# B&R Automation Studio project NAINV104C00R8L515F00 (part 21)

#### Act_Link.st - Change By Project
```iecst
(** 2019-03-29 **)
ACTION Act_Link:

	//Ready Receive
	IF p_bLinkNtParamUSWidthChkPrep AND p_bLinkMcParamUSWidthChkEn THEN
		p_bRdyRcv	:= p_bLinkDIUSWidthChkSen;
	ELSE
		p_bRdyRcv	:= TRUE;
	END_IF

	//Receive Complete Signal
	//p_bComplSigOn	:= p_bLeftSen = FALSE;

	IF EDGENEG(p_bLeftSen) THEN
		p_bComplSigOn	:= TRUE;
	END_IF

	IF eStat <> SMEMAActRun THEN
		p_bComplSigOn	:= FALSE;
	END_IF

	//Direction
	p_bDirLToR	:= p_eLinkConvDir = ConvDirLToR OR p_eLinkConvDir = ConvDirLToL;

END_ACTION
```

#### Act_InitLocal.st - Do Not Change!!!
```iecst
(** 2019-03-25 **)
ACTION Act_InitLocal:

	//Input Reference Link To Local Variable
	p_eAct ACCESS ADR(eAct);
	p_udiRstErr ACCESS ADR(udiRstErr);
	p_bPrep ACCESS ADR(bPrep);
	p_bEn ACCESS ADR(bEn);
	p_bDis ACCESS ADR(bDis);
	p_bManual ACCESS ADR(bManual);
	p_tyParam ACCESS ADR(tyParam);
	p_diTransferInTO ACCESS ADR(diTransferInTO);
	p_bDirLToR ACCESS ADR(bDirLToR);
	p_bRdyRcv ACCESS ADR(bRdyRcv);
	p_bLeftSen ACCESS ADR(bLeftSen);
	p_bRightSen ACCESS ADR(bRightSen);
	p_bComplSigOn ACCESS ADR(bComplSigOn);
	p_bUBA ACCESS ADR(bUBA);
	p_bUBAStat ACCESS ADR(bUBAStat);
	p_bTimerEnSen ACCESS ADR(bTimerEnSen);
	p_bTimerEnSenEdge ACCESS ADR(bTimerEnSenEdge);
	p_bVirtualEn ACCESS ADR(bVirtualEn);
	p_bUBAVirtual ACCESS ADR(bUBAVirtual);
	p_bUBAStatVirtual ACCESS ADR(bUBAStatVirtual);
	p_tRstDlyTm ACCESS ADR(tRstDlyTm);
	p_tSigInChkTm ACCESS ADR(tSigInChkTm);
	p_sProgNm ACCESS ADR(sProgNm);
	p_bNtSettingsLoadDone ACCESS ADR(bNtSettingsLoadDone);

END_ACTION
```

#### Act_Initial.st - Do Not Change!!!
```iecst
(** 2019-03-22 **)
ACTION Act_Initial:

	//Initial
	sStatTxt	:= a_sStatText[eStat];

	fbSMEMA_Std.tRstDlyTm	:= p_tRstDlyTm;
	fbSMEMA_Std(bEn := FALSE);

	fbSMEMA_9851.tRstDlyTm	:= p_tRstDlyTm;
	fbSMEMA_9851(bEn := FALSE);

	fbTimerDlyTm(IN := FALSE);
	fbTimeTrig(CLK := TRUE);

	fbSigInChk.tSigInChkTm	:= p_tSigInChkTm;

END_ACTION
```

#### Act_Background.st - Do Not Change!!!
```iecst
(** 2019-01-20 **)
ACTION Act_Background:

	fbTimeTrig(CLK := p_bTimerEnSenEdge);

	IF eStat = SMEMAActRun AND (p_bTimerEnSenEdge OR p_bTimerEnSen) THEN
		IF fbTimeTrig.Q = TRUE OR p_bTimerEnSen THEN
			fbTimerDlyTm.IN	:= TRUE;
		END_IF
	ELSE
		fbTimerDlyTm.IN	:= FALSE;
	END_IF

	IF bConvStart = FALSE AND bConvStop = FALSE THEN
		fbTimerDlyTm;

		IF fbTimerDlyTm.Q = TRUE AND eStat = SMEMAActRun THEN
			bTimer		:= TRUE;
			bVirtual	:= FALSE;
		ELSIF p_bVirtualEn = TRUE THEN
			bTimer		:= FALSE;
			bVirtual	:= TRUE;
		ELSE
			bTimer		:= FALSE;
			bVirtual	:= FALSE;
		END_IF
	ELSE
		fbTimerDlyTm(IN := FALSE);
	END_IF

	IF bTimer = TRUE THEN

		fbSigInChk.bNomSig			:= bConvStart = FALSE AND bConvStop = FALSE;
		fbSigInChk.bStatSig			:= FALSE;
		fbSigInChk.bStatSigSetGd	:= FALSE;

	ELSIF bVirtual = TRUE THEN

		fbSigInChk.bNomSig	:= p_bUBAVirtual;

		IF p_tyParam.eSelection = SMEMASelIPC9851Ext THEN
			fbSigInChk.bStatSig			:= p_bUBAStatVirtual;
			fbSigInChk.bStatSigSetGd	:= p_tyParam.bStatSigSetGd;
		ELSE
			fbSigInChk.bStatSig			:= FALSE;
			fbSigInChk.bStatSigSetGd	:= FALSE;
		END_IF

	ELSE

		fbSigInChk.bNomSig	:= p_bUBA;

		IF p_tyParam.eSelection = SMEMASelIPC9851Ext THEN
			fbSigInChk.bStatSig			:= p_bUBAStat;
			fbSigInChk.bStatSigSetGd	:= p_tyParam.bStatSigSetGd;
		ELSE
			fbSigInChk.bStatSig			:= FALSE;
			fbSigInChk.bStatSigSetGd	:= FALSE;
		END_IF

	END_IF

	fbSigInChk;

	bUSRdy		:= fbSigInChk.bSigInValid;
	bUSGdBrdRdy	:= fbSigInChk.bGdBrd;

END_ACTION
```

#### InputRef.var - Do Not Change!!!
```iecst
(*2019-03-25*)
(**)
(*General*)
VAR
	p_eAct : REFERENCE TO eSMEMAAction;
	p_udiRstErr : REFERENCE TO UDINT;
	p_bPrep : REFERENCE TO BOOL;
	p_bEn : REFERENCE TO BOOL;
	p_bDis : REFERENCE TO BOOL;
END_VAR
(**)
(*Configuration*)
VAR
	p_bManual : REFERENCE TO BOOL;
	p_tyParam : REFERENCE TO tySMEMAParam;
	p_diTransferInTO : REFERENCE TO DINT;
	p_bDirLToR : REFERENCE TO BOOL;
	p_bRdyRcv : REFERENCE TO BOOL;
END_VAR
(**)
(*Input*)
VAR
	p_bLeftSen : REFERENCE TO BOOL;
	p_bRightSen : REFERENCE TO BOOL;
	p_bComplSigOn : REFERENCE TO BOOL;
	p_bUBA : REFERENCE TO BOOL;
	p_bUBAStat : REFERENCE TO BOOL;
	p_bTimerEnSen : REFERENCE TO BOOL;
	p_bTimerEnSenEdge : REFERENCE TO BOOL;
	p_bVirtualEn : REFERENCE TO BOOL;
	p_bUBAVirtual : REFERENCE TO BOOL;
	p_bUBAStatVirtual : REFERENCE TO BOOL;
	p_tRstDlyTm : REFERENCE TO TIME;
	p_tSigInChkTm : REFERENCE TO TIME;
	p_sProgNm : REFERENCE TO STRING[15];
	p_bNtSettingsLoadDone : REFERENCE TO BOOL;
END_VAR
```

#### Local.var - Do Not Change!!!
```iecst
(*2019-04-30*)
(**)
(*Local Action, State & Status*)
VAR
	eAct : eSMEMAAction := SMEMAActIdle;
	eStat : eSMEMAAction := SMEMAActIdle;
	eStatus : eFBStatus := Idle;
	udiStatus : UDINT := 0;
	sStatTxt : STRING[200] := '';
	a_sStatText : ARRAY[0..50] OF STRING[200] := ['Idling','Upstream SMEMA Running','Turning On USB Signal','NA','Turning Off USB Signal','NA','Turning On USB Signal','Turning Off USB Signal',43('')];
END_VAR
(**)
(*Local Alarm*)
VAR
	tyAlmData : tyAlmDat;
	a_tyAlmText : ARRAY[10000..10099] OF tyAlmTxt := [(sAlmText:='SMEMA 9851 Transport Time Out While Transporting',sRcyText:='Timeout Expired Before Operation Completed. Reset And Resume Operation.'),(sAlmText:='SMEMA 9851 Transport Time Out After Opposite Machine Transport Finished',sRcyText:='Timeout Expired Before Operation Completed. Reset And Resume Operation.'),(sAlmText:='SMEMA 9851 Transport Time Out After Current Machine Transport Finished',sRcyText:='Timeout Expired Before Operation Completed. Reset And Resume Operation.'),(sAlmText:='SMEMA 9851 Transport Time Out After Both Machine Transport Finished And Waiting Outlet Sensor',sRcyText:='Timeout Expired Before Operation Completed. Reset And Resume Operation.'),(sAlmText:='Standard SMEMA Transport Time Out While Transporting',sRcyText:='Timeout Expired Before Operation Completed. Reset And Resume Operation.'),(sAlmText:='Standard SMEMA Transport Time Out After Opposite Machine Transport Finished',sRcyText:='Timeout Expired Before Operation Completed. Reset And Resume Operation.'),(sAlmText:='Standard SMEMA Transport Time Out After Current Machine Transport Finished',sRcyText:='Timeout Expired Before Operation Completed. Reset And Resume Operation.'),(sAlmText:='Standard SMEMA Transport Time Out After Both Machine Transport Finished And Waiting Outlet Sensor',sRcyText:='Timeout Expired Before Operation Completed. Reset And Resume Operation.'),92((0))];
END_VAR
(**)
(*Local Output*)
VAR
	bUSRdy : BOOL := FALSE;
	bUSGdBrdRdy : BOOL := FALSE;
	bDSRdy : BOOL := FALSE;
	bTransporting : BOOL := FALSE;
	bConvStart : BOOL := FALSE;
	bConvStop : BOOL := FALSE;
	bUSB : BOOL := FALSE;
	bTimer : BOOL;
	bVirtual : BOOL;
END_VAR
(**)
(*Local Input*)
VAR
	udiRstErr : UDINT := 0;
	bPrep : BOOL := TRUE;
	bEn : BOOL := TRUE;
	bDis : BOOL := FALSE;
	bManual : BOOL := FALSE;
	tyParam : tySMEMAParam;
	diTransferInTO : DINT := 20000;
	bDirLToR : BOOL := FALSE;
	bRdyRcv : BOOL := TRUE;
	bLeftSen : BOOL := FALSE;
	bRightSen : BOOL := FALSE;
	bComplSigOn : BOOL := FALSE;
	bUBA : BOOL := FALSE;
	bUBAStat : BOOL := FALSE;
	bTimerEnSen : BOOL;
	bTimerEnSenEdge : BOOL;
	bVirtualEn : BOOL;
	bUBAVirtual : BOOL;
	bUBAStatVirtual : BOOL;
	tRstDlyTm : TIME := T#500ms;
	tSigInChkTm : TIME := T#100ms;
	sProgNm : STRING[15] := 'USSMEMA';
	bNtSettingsLoadDone : BOOL := TRUE;
END_VAR
(**)
(*Local*)
VAR
	bRstErr : BOOL;
	udiRstErrOld : UDINT;
	bInitDone : BOOL;
	bInitialDone : BOOL;
	fbTimerDlyTm : TON := (PT:=T#1s);
	fbTimeTrig : R_TRIG;
	fbSMEMA_Std : fbSMEMAUS_Std;
	fbSMEMA_9851 : fbSMEMAUS_9851;
	fbSigInChk : fbSMEMASigInChk;
	eStatOld : eSMEMAAction := SMEMAActIdle;
	udiModuleNum : UDINT := 2701;
END_VAR
```

### DSSMEMA.var - Change By Project
```iecst
(*2019-03-25*)
(**)
(*Action & State & Status*)
VAR
	p_DSSMEMAStat : UDINT;
	p_DSSMEMAStatus : UDINT;
	p_DSSMEMAStatTxt : UDINT;
END_VAR
(**)
(*Alarm*)
VAR
	p_DSSMEMAAlmData : UDINT;
END_VAR
(**)
(*Output*)
VAR
	p_DSSMEMAUSRdy : UDINT;
	p_DSSMEMAUSGdBrdRdy : UDINT;
	p_DSSMEMADSRdy : UDINT;
	p_DSSMEMATransporting : UDINT;
	p_DSSMEMAConvStart : UDINT;
	p_DSSMEMAConvStop : UDINT;
	p_DSSMEMADBA : UDINT;
	p_DSSMEMADBAStat : UDINT;
	p_DSSMEMATimer : UDINT;
	p_DSSMEMAVirtual : UDINT;
END_VAR
```

### Program Logical/SMEMA/DSSMEMA (IEC) - 1.00.0 - NtSMEMA v5.00.0

#### InputRef.var
```iecst
(*2019-03-25*)
(**)
(*General*)
VAR
	p_eAct : REFERENCE TO eSMEMAAction;
	p_udiRstErr : REFERENCE TO UDINT;
	p_bPrep : REFERENCE TO BOOL;
	p_bEn : REFERENCE TO BOOL;
	p_bDis : REFERENCE TO BOOL;
END_VAR
(**)
(*Configuration*)
VAR
	p_bManual : REFERENCE TO BOOL;
	p_tyParam : REFERENCE TO tySMEMAParam;
	p_bGdBrd : REFERENCE TO BOOL;
	p_diTransferOutTO : REFERENCE TO DINT;
	p_bDirLToR : REFERENCE TO BOOL;
	p_bRdySend : REFERENCE TO BOOL;
END_VAR
(**)
(*Input*)
VAR
	p_bLeftSen : REFERENCE TO BOOL;
	p_bRightSen : REFERENCE TO BOOL;
	p_bComplSigOn : REFERENCE TO BOOL;
	p_bDSB : REFERENCE TO BOOL;
	p_bTimerEnSen : REFERENCE TO BOOL;
	p_bTimerEnSenEdge : REFERENCE TO BOOL;
	p_bVirtualEn : REFERENCE TO BOOL;
	p_bDSBVirtual : REFERENCE TO BOOL;
	p_tRstDlyTm : REFERENCE TO TIME;
	p_tSigInChkTm : REFERENCE TO TIME;
	p_sProgNm : REFERENCE TO STRING[15];
	p_bNtSettingsLoadDone : REFERENCE TO BOOL;
END_VAR
```

#### InputRef_Link.var
```iecst
(*2019-04-09*)
(**)
VAR
	p_bLinkOpsRun : REFERENCE TO BOOL;
END_VAR
(**)
VAR
	p_eLinkConvDir : REFERENCE TO eConvDir;
	p_bLinkNtParamDSWidthChkPrep : REFERENCE TO BOOL;
	p_bLinkMcParamDSWidthChkEn : REFERENCE TO BOOL;
	p_bLinkDIDSWidthChkSen : REFERENCE TO BOOL;
	p_usiLinkMcMod : REFERENCE TO USINT;
END_VAR
```

#### Local.var
```iecst
(*2019-04-30*)
(**)
(*Local Action, State & Status*)
VAR
	eAct : eSMEMAAction := SMEMAActIdle;
	eStat : eSMEMAAction := SMEMAActIdle;
	eStatus : eFBStatus := Idle;
	udiStatus : UDINT := 0;
	sStatTxt : STRING[200] := '';
	a_sStatText : ARRAY[0..50] OF STRING[200] := ['Idling','SMEMA Running','Turning On DBA Signal','Turning On DBA Stat Signal','Turning Off DBA Signal','Turning Off DBA Stat Signal','Turning On All DBA Signal','Turning Off All DBA Signal',43('')];
END_VAR
(**)
(*Local Alarm*)
VAR
	tyAlmData : tyAlmDat;
	a_tyAlmText : ARRAY[10000..10099] OF tyAlmTxt := [(sAlmText:='SMEMA 9851 Transport Time Out While Transporting',sRcyText:='Timeout Expired Before Operation Completed. Reset And Resume Operation.'),(sAlmText:='SMEMA 9851 Transport Time Out After Opposite Machine Transport Finished',sRcyText:='Timeout Expired Before Operation Completed. Reset And Resume Operation.'),(sAlmText:='SMEMA 9851 Transport Time Out After Current Machine Transport Finished',sRcyText:='Timeout Expired Before Operation Completed. Reset And Resume Operation.'),(sAlmText:='SMEMA 9851 Transport Time Out After Both Machine Transport Finished And Waiting Outlet Sensor',sRcyText:='Timeout Expired Before Operation Completed. Reset And Resume Operation.'),(sAlmText:='Standard SMEMA Transport Time Out While Transporting',sRcyText:='Timeout Expired Before Operation Completed. Reset And Resume Operation.'),(sAlmText:='Standard SMEMA Transport Time Out After Opposite Machine Transport Finished',sRcyText:='Timeout Expired Before Operation Completed. Reset And Resume Operation.'),(sAlmText:='Standard SMEMA Transport Time Out After Current Machine Transport Finished',sRcyText:='Timeout Expired Before Operation Completed. Reset And Resume Operation.'),(sAlmText:='Standard SMEMA Transport Time Out After Both Machine Transport Finished And Waiting Outlet Sensor',sRcyText:='Timeout Expired Before Operation Completed. Reset And Resume Operation.'),92((0))];
END_VAR
(**)
(*Local Output*)
VAR
	bUSRdy : BOOL := FALSE;
	bUSGdBrdRdy : BOOL := FALSE;
	bDSRdy : BOOL := FALSE;
	bTransporting : BOOL := FALSE;
	bConvStart : BOOL := FALSE;
	bConvStop : BOOL := FALSE;
	bDBA : BOOL := FALSE;
	bDBAStat : BOOL := FALSE;
	bTimer : BOOL;
	bVirtual : BOOL;
END_VAR
(**)
(*Local Input*)
VAR
	udiRstErr : UDINT := 0;
	bPrep : BOOL := TRUE;
	bEn : BOOL := TRUE;
	bDis : BOOL := FALSE;
	bManual : BOOL := FALSE;
	tyParam : tySMEMAParam;
	bGdBrd : BOOL := TRUE;
	diTransferOutTO : DINT := 20000;
	bDirLToR : BOOL := FALSE;
	bRdySend : BOOL := TRUE;
	bLeftSen : BOOL := FALSE;
	bRightSen : BOOL := FALSE;
	bComplSigOn : BOOL := FALSE;
	bDSB : BOOL := FALSE;
	bTimerEnSen : BOOL;
	bTimerEnSenEdge : BOOL;
	bVirtualEn : BOOL;
	bDSBVirtual : BOOL;
	tRstDlyTm : TIME := T#500ms;
	tSigInChkTm : TIME := T#100ms;
	sProgNm : STRING[15] := 'DSSMEMA';
	bNtSettingsLoadDone : BOOL := TRUE;
END_VAR
(**)
(*Local*)
VAR
	bRstErr : BOOL;
	udiRstErrOld : UDINT;
	bInitDone : BOOL;
	bInitialDone : BOOL;
	fbTimerDlyTm : TON := (PT:=T#1s);
	fbTimeTrig : R_TRIG;
	fbSMEMA_OppFirst : fbSMEMADS_OppFirst;
	fbSMEMA : fbSMEMADS;
	fbSigInChk : fbSMEMASigInChk;
	eStatOld : eSMEMAAction := SMEMAActIdle;
	udiModuleNum : UDINT := 2801;
END_VAR
```

#### Act_Action.st
```iecst
(** 2019-03-25 **)
ACTION Act_Action:

	//Reset Error
	IF (eStatus = Error) AND bRstErr THEN
		p_eAct	:= SMEMAActIdle;
		eStat	:= SMEMAActIdle;
	END_IF

	//Set p_eAct
	IF eStatus = Idle OR eStatus = Busy OR eStatus = Done THEN
		eStat	:= p_eAct;
	END_IF

END_ACTION
```

#### Act_Alarm.st
```iecst
(** 2019-03-25 **)
ACTION Act_Alarm:

	//Error
	IF EDGEPOS(eStatus = Error) THEN

		tyAlmData.sProgNm		:= p_sProgNm;
		tyAlmData.udiCode		:= udiStatus;
		tyAlmData.eSeverity		:= AlmSeverityError;
		tyAlmData.udiRunTime	:= tyAlmData.udiRunTime + 1;
		tyAlmData.bAlm			:= TRUE;
		tyAlmData.udiModuleNum  := udiModuleNum;
		g_sDSSMEMAProgNm		:= p_sProgNm;

		//Get Error Message
		IF tyAlmData.udiCode < 10000 OR tyAlmData.udiCode > 10099 THEN
			tyAlmData.sAlmMsg	:= 'Unknown';
			tyAlmData.sRcyMsg	:= 'Unknown';
		ELSE
			tyAlmData.sAlmMsg	:= a_tyAlmText[tyAlmData.udiCode].sAlmText;
			tyAlmData.sRcyMsg	:= a_tyAlmText[tyAlmData.udiCode].sRcyText;
		END_IF

		sStatTxt	:= tyAlmData.sAlmMsg;

	ELSIF bRstErr AND (tyAlmData.udiCode <> 0) THEN

		tyAlmData.udiCode	:= 0;
		tyAlmData.eSeverity	:= AlmSeverityNA;
		tyAlmData.sAlmMsg	:= '';
		tyAlmData.sRcyMsg	:= '';
		tyAlmData.bAlm			:= FALSE;
		sStatTxt	:= a_sStatText[eStat];

	END_IF

END_ACTION
```

#### Act_Background.st
```iecst
(** 2019-01-20 **)
ACTION Act_Background:

	fbTimeTrig(CLK := p_bTimerEnSenEdge);

	IF eStat = SMEMAActRun AND (p_bTimerEnSenEdge OR p_bTimerEnSen) THEN
		IF fbTimeTrig.Q = TRUE OR p_bTimerEnSen THEN
			fbTimerDlyTm.IN	:= TRUE;
		END_IF
	ELSE
		fbTimerDlyTm.IN	:= FALSE;
	END_IF

	IF bConvStart = FALSE AND bConvStop = FALSE THEN
		fbTimerDlyTm;

		IF fbTimerDlyTm.Q = TRUE AND eStat = SMEMAActRun THEN
			bTimer		:= TRUE;
			bVirtual	:= FALSE;
		ELSIF p_bVirtualEn = TRUE THEN
			bTimer		:= FALSE;
			bVirtual	:= TRUE;
		ELSE
			bTimer		:= FALSE;
			bVirtual	:= FALSE;
		END_IF
	ELSE
		fbTimerDlyTm(IN := FALSE);
	END_IF

	IF bTimer = TRUE THEN

		fbSigInChk.bNomSig			:= bConvStart = FALSE AND bConvStop = FALSE;
		fbSigInChk.bStatSig			:= FALSE;
		fbSigInChk.bStatSigSetGd	:= FALSE;

	ELSIF bVirtual = TRUE THEN

		fbSigInChk.bNomSig			:= p_bDSBVirtual;
		fbSigInChk.bStatSig			:= FALSE;
		fbSigInChk.bStatSigSetGd	:= FALSE;

	ELSE

		fbSigInChk.bNomSig			:= p_bDSB;
		fbSigInChk.bStatSig			:= FALSE;
		fbSigInChk.bStatSigSetGd	:= FALSE;

	END_IF

	fbSigInChk;

	bDSRdy	:= fbSigInChk.bSigInValid;

END_ACTION
```

#### Act_InitGlobal.st
```iecst
(** 2019-04-09 **)
ACTION Act_InitGlobal:

	(* Always Change If Project Change *)

	//Pass Data To Link
	p_bLinkOpsRun ACCESS p_OpsRun;

	p_eLinkConvDir ACCESS p_NtParamProjConvDir;
	p_bLinkNtParamDSWidthChkPrep ACCESS p_NtParamDSWidthChkPrep;
	p_bLinkMcParamDSWidthChkEn ACCESS p_McParamDSWidthChkEn;
	p_bLinkDIDSWidthChkSen ACCESS p_DIDSWidthChkSen;

	p_usiLinkMcMod ACCESS p_ProdRcpCurrRcp0McMod;

	//Pass Data To Internal Use
	p_udiRstErr ACCESS p_RstErrReset;
	p_bManual ACCESS p_UIMnlMod;
	p_tyParam ACCESS p_McParamDSSMEMAParam;
	p_diTransferOutTO ACCESS p_McParamTranOutErrDlyTm;
	p_bLeftSen ACCESS p_DIConvLftSen;
	p_bRightSen ACCESS p_DIConvRgtSen;
	p_bDSB ACCESS p_DIDSB;
	p_bVirtualEn ACCESS p_UIVSMEMADSEn;
	p_bDSBVirtual ACCESS p_UIVSMEMADSB;
	p_tRstDlyTm ACCESS p_NtParamDSSMEMARstDlyTm;
	p_tSigInChkTm ACCESS p_NtParamDSSMEMASigInChkTm;
	p_sProgNm ACCESS p_NtParamDSSMEMAProgNm;
	p_bNtSettingsLoadDone ACCESS p_StartupNtSettingsLoadDone;

//	p_bGdBrd ACCESS p_OpsInvertGdBrd;

	(* Always Change If Project Change *)

END_ACTION
```

#### Act_Initial.st
```iecst
(** 2019-04-27 **)
ACTION Act_Initial:

	//Initial
	sStatTxt	:= a_sStatText[eStat];

	fbSMEMA_OppFirst.tRstDlyTm	:= p_tRstDlyTm;
	fbSMEMA_OppFirst(bEn := FALSE);

	fbSMEMA.tRstDlyTm	:= p_tRstDlyTm;
	fbSMEMA(bEn := FALSE);

	fbTimerDlyTm(IN := FALSE);
	fbTimeTrig(CLK := TRUE);

	fbSigInChk.tSigInChkTm	:= p_tSigInChkTm;

END_ACTION
```

#### Act_InitLocal.st
```iecst
(** 2019-03-25 **)
ACTION Act_InitLocal:

	//Input Reference Link To Local Variable
	p_eAct ACCESS ADR(eAct);
	p_udiRstErr ACCESS ADR(udiRstErr);
	p_bPrep ACCESS ADR(bPrep);
	p_bEn ACCESS ADR(bEn);
	p_bDis ACCESS ADR(bDis);
	p_bManual ACCESS ADR(bManual);
	p_tyParam ACCESS ADR(tyParam);
	p_bGdBrd ACCESS ADR(bGdBrd);
	p_diTransferOutTO ACCESS ADR(diTransferOutTO);
	p_bDirLToR ACCESS ADR(bDirLToR);
	p_bRdySend ACCESS ADR(bRdySend);
	p_bLeftSen ACCESS ADR(bLeftSen);
	p_bRightSen ACCESS ADR(bRightSen);
	p_bComplSigOn ACCESS ADR(bComplSigOn);
	p_bDSB ACCESS ADR(bDSB);
	p_bTimerEnSen ACCESS ADR(bTimerEnSen);
	p_bTimerEnSenEdge ACCESS ADR(bTimerEnSenEdge);
	p_bVirtualEn ACCESS ADR(bVirtualEn);
	p_bDSBVirtual ACCESS ADR(bDSBVirtual);
	p_tRstDlyTm ACCESS ADR(tRstDlyTm);
	p_tSigInChkTm ACCESS ADR(tSigInChkTm);
	p_sProgNm ACCESS ADR(sProgNm);
	p_bNtSettingsLoadDone ACCESS ADR(bNtSettingsLoadDone);

END_ACTION
```

#### Act_Link.st
```iecst
(** 2019-03-29 **)
ACTION Act_Link:

	//Ready Send
	IF p_bLinkNtParamDSWidthChkPrep AND p_bLinkMcParamDSWidthChkEn THEN
		p_bRdySend	:= p_bLinkDIDSWidthChkSen;
	ELSE
		p_bRdySend	:= TRUE;
	END_IF

	//Send Complete Signal
	IF EDGENEG(p_bRightSen) THEN
		p_bComplSigOn	:= TRUE;
	END_IF

	IF eStat <> SMEMAActRun THEN
		p_bComplSigOn	:= FALSE;
	END_IF

	//Direction
	p_bDirLToR	:= p_eLinkConvDir = ConvDirLToR OR p_eLinkConvDir = ConvDirLToL;

	//Good Board Access
	IF p_usiLinkMcMod = 0 AND p_usiLinkMcMod = 1 THEN
		p_bGdBrd ACCESS p_OpsInvertGdBrd;
	ELSE
		p_bGdBrd ACCESS p_OpsInvertGdBrd;
	END_IF

END_ACTION
```

#### Act_LinkAction.st
```iecst
(** 2019-04-09 **)
ACTION Act_LinkAction:

	IF p_bLinkOpsRun = TRUE THEN
		p_eAct ACCESS p_OpsInvertDSSMEMAAct;
	ELSIF p_bManual = TRUE THEN
		p_eAct ACCESS p_UIDSSMEMAAct;
	ELSE
		p_eAct ACCESS ADR(eAct);
	END_IF

END_ACTION
```

#### Act_Main.st
```iecst
(** 2019-04-27 **)
ACTION Act_Main:

	IF eStatOld <> eStat THEN
		fbSMEMA_OppFirst(bEn := FALSE);
		fbSMEMA(bEn := FALSE);

		bTransporting	:= FALSE;
		bConvStart		:= FALSE;
		bConvStop		:= FALSE;
		bUSRdy			:= FALSE;
		bUSGdBrdRdy		:= FALSE;

		IF eStatOld <> SMEMAActIdle
			AND eStatOld <> SMEMAActSetSig
			AND eStatOld <> SMEMAActSetStatSig
			AND eStatOld <> SMEMAActRstSig
			AND eStatOld <> SMEMAActRstStatSig
			AND eStatOld <> SMEMAActSetAllSig
			AND eStatOld <> SMEMAActRstAllSig THEN

			bDBA		:= FALSE;
			bDBAStat	:= FALSE;

		END_IF

		sStatTxt	:= a_sStatText[eStat];

		eStatOld	:= eStat;

		eStatus		:= Busy;
	END_IF

	//Main
	CASE eStat OF

		SMEMAActIdle:
			IF EDGENEG(p_bManual) THEN
				bDBA		:= FALSE;
				bDBAStat	:= FALSE;
			END_IF

			eStatus	:= Idle;

		SMEMAActRun:
			IF eStatus = Idle OR eStatus = Busy THEN

				eStatus	:= Busy;

				IF p_tyParam.eSelection <> SMEMASelStandard THEN

					fbSMEMA.bDSRdy		:= fbSigInChk.bSigInValid;
					fbSMEMA.bRdySend	:= p_bRdySend;
					fbSMEMA.bComplSigOn	:= p_bComplSigOn;

					fbSMEMA.tTimeOut	:= DINT_TO_TIME(p_diTransferOutTO);
					fbSMEMA(bEn := TRUE);

					bTransporting	:= fbSMEMA.bTransporting;
					bConvStart		:= fbSMEMA.bConvStart;
					bConvStop		:= fbSMEMA.bConvStop;
					bDBA			:= fbSMEMA.bSigToDS AND (bTimer = FALSE) AND (bVirtual = FALSE);
					bDBAStat		:= (fbSMEMA.bSigToDS) AND (fSMEMASigStatOut(p_tyParam.bStatSigSetGd, p_bGdBrd)) AND (p_tyParam.eSelection = SMEMASelIPC9851Ext);

					bUSRdy			:= fbSMEMA.bSigToDS;
					bUSGdBrdRdy		:= p_bGdBrd;

					IF fbSMEMA.udiStatus = 0 THEN
						eStatus	:= Done;
					ELSIF fbSMEMA.udiStatus < 65534 THEN
						eStatus		:= Error;

						IF fbSMEMA.udiStatus = 1200 THEN
							udiStatus	:= 10000;	//SMEMA 9851 Transport Time Out While Transporting
						ELSIF fbSMEMA.udiStatus = 1201 THEN
							udiStatus	:= 10001;	//SMEMA 9851 Transport Time Out After Opposite Machine Transport Finished
						ELSIF fbSMEMA.udiStatus = 1202 THEN
							udiStatus	:= 10002;	//SMEMA 9851 Transport Time Out After Current Machine Transport Finished
						ELSIF fbSMEMA.udiStatus = 1203 THEN
							udiStatus	:= 10003;	//SMEMA 9851 Transport Time Out After Both Machine Transport Finished And Waiting Outlet Sensor
						ELSE
							udiStatus	:= fbSMEMA.udiStatus;
						END_IF
					END_IF

				ELSE

					fbSMEMA_OppFirst.bDSRdy			:= fbSigInChk.bSigInValid;
					fbSMEMA_OppFirst.bRdySend		:= p_bRdySend;
					fbSMEMA_OppFirst.bComplSigOn	:= p_bComplSigOn;

					fbSMEMA_OppFirst.tTimeOut	:= DINT_TO_TIME(p_diTransferOutTO);
					fbSMEMA_OppFirst(bEn := TRUE);

					bTransporting	:= fbSMEMA_OppFirst.bTransporting;
					bConvStart		:= fbSMEMA_OppFirst.bConvStart;
					bConvStop		:= fbSMEMA_OppFirst.bConvStop;
					bDBA			:= fbSMEMA_OppFirst.bSigToDS AND (bTimer = FALSE) AND (bVirtual = FALSE);
					bDBAStat		:= (fbSMEMA_OppFirst.bSigToDS) AND (fSMEMASigStatOut(p_tyParam.bStatSigSetGd, p_bGdBrd)) AND (p_tyParam.eSelection = SMEMASelIPC9851Ext);

					bUSRdy			:= fbSMEMA_OppFirst.bSigToDS;
					bUSGdBrdRdy		:= p_bGdBrd;

					IF fbSMEMA_OppFirst.udiStatus = 0 THEN
						eStatus	:= Done;
					ELSIF fbSMEMA_OppFirst.udiStatus < 65534 THEN
						eStatus		:= Error;

						IF fbSMEMA_OppFirst.udiStatus = 1200 THEN
							udiStatus	:= 10004;	//Standard SMEMA Transport Time Out While Transporting
						ELSIF fbSMEMA_OppFirst.udiStatus = 1201 THEN
							udiStatus	:= 10005;	//Standard SMEMA Transport Time Out After Opposite Machine Transport Finished
						ELSIF fbSMEMA_OppFirst.udiStatus = 1202 THEN
							udiStatus	:= 10006;	//Standard SMEMA Transport Time Out After Current Machine Transport Finished
						ELSIF fbSMEMA_OppFirst.udiStatus = 1203 THEN
							udiStatus	:= 10007;	//Standard SMEMA Transport Time Out After Both Machine Transport Finished And Waiting Outlet Sensor
						ELSE
							udiStatus	:= fbSMEMA_OppFirst.udiStatus;
						END_IF
					END_IF

				END_IF

			END_IF

		SMEMAActSetSig:
			IF eStatus = Idle OR eStatus = Busy THEN

				//Reset
				fbSMEMA_OppFirst(bEn := FALSE);
				fbSMEMA(bEn := FALSE);

				bConvStart	:= FALSE;
				bConvStop	:= FALSE;

				bDBA	:= TRUE;
				eStatus	:= Done;

			END_IF

		SMEMAActSetStatSig:
			IF eStatus = Idle OR eStatus = Busy THEN

				//Reset
				fbSMEMA_OppFirst(bEn := FALSE);
				fbSMEMA(bEn := FALSE);

				bConvStart	:= FALSE;
				bConvStop	:= FALSE;

				bDBAStat	:= TRUE;
				eStatus		:= Done;

			END_IF

		SMEMAActRstSig:
			IF eStatus = Idle OR eStatus = Busy THEN

				//Reset
				fbSMEMA_OppFirst(bEn := FALSE);
				fbSMEMA(bEn := FALSE);

				bConvStart	:= FALSE;
				bConvStop	:= FALSE;

				bDBA	:= FALSE;
				eStatus	:= Done;

			END_IF

		SMEMAActRstStatSig:
			IF eStatus = Idle OR eStatus = Busy THEN

				//Reset
				fbSMEMA_OppFirst(bEn := FALSE);
				fbSMEMA(bEn := FALSE);

				bConvStart	:= FALSE;
				bConvStop	:= FALSE;

				bDBAStat	:= FALSE;
				eStatus		:= Done;

			END_IF

		SMEMAActSetAllSig:
			IF eStatus = Idle OR eStatus = Busy THEN

				//Reset
				fbSMEMA_OppFirst(bEn := FALSE);
				fbSMEMA(bEn := FALSE);

				bConvStart	:= FALSE;
				bConvStop	:= FALSE;

				bDBA		:= TRUE;
				bDBAStat	:= TRUE;
				eStatus		:= Done;

			END_IF

		SMEMAActRstAllSig:
			IF eStatus = Idle OR eStatus = Busy THEN

				//Reset
				fbSMEMA_OppFirst(bEn := FALSE);
				fbSMEMA(bEn := FALSE);

				bConvStart	:= FALSE;
				bConvStop	:= FALSE;

				bDBA		:= FALSE;
				bDBAStat	:= FALSE;
				eStatus		:= Done;

			END_IF

	END_CASE

END_ACTION
```

#### Init.st
```iecst
(** 2019-03-25 **)
PROGRAM _INIT

	(* Always Change If Project Change *)

	//Pass Address To Global Address For External Use
	//Action, State & Status
	p_DSSMEMAStat		:= ADR(eStat);
	p_DSSMEMAStatus		:= ADR(eStatus);
	p_DSSMEMAStatTxt	:= ADR(sStatTxt);

	//Alarm
	p_DSSMEMAAlmData	:= ADR(tyAlmData);

	//Output
	p_DSSMEMAUSRdy			:= ADR(bUSRdy);
	p_DSSMEMAUSGdBrdRdy		:= ADR(bUSGdBrdRdy);
	p_DSSMEMADSRdy			:= ADR(bDSRdy);
	p_DSSMEMATransporting	:= ADR(bTransporting);
	p_DSSMEMAConvStart		:= ADR(bConvStart);
	p_DSSMEMAConvStop		:= ADR(bConvStop);
	p_DSSMEMADBA			:= ADR(bDBA);
	p_DSSMEMADBAStat		:= ADR(bDBAStat);
	p_DSSMEMATimer			:= ADR(bTimer);
	p_DSSMEMAVirtual		:= ADR(bVirtual);

	(* Always Change If Project Change *)

END_PROGRAM
```

### USSMEMA2.var - Change By Project
```iecst
(*2019-03-25*)
(**)
(*Action & State & Status*)
VAR
	p_USSMEMA2Stat : UDINT;
	p_USSMEMA2Status : UDINT;
	p_USSMEMA2StatTxt : UDINT;
END_VAR
(**)
(*Alarm*)
VAR
	p_USSMEMA2AlmData : UDINT;
END_VAR
(**)
(*Output*)
VAR
	p_USSMEMA2USRdy : UDINT;
	p_USSMEMA2USGdBrdRdy : UDINT;
	p_USSMEMA2DSRdy : UDINT;
	p_USSMEMA2Transporting : UDINT;
	p_USSMEMA2ConvStart : UDINT;
	p_USSMEMA2ConvStop : UDINT;
	p_USSMEMA2USB : UDINT;
	p_USSMEMA2Timer : UDINT;
	p_USSMEMA2Virtual : UDINT;
END_VAR
```

### Program Logical/SMEMA/USSMEMA2 (IEC, version 1.00.0) - 1.00.0 - NtSMEMA v5.00.0

#### Init.st - Change By Project
```iecst
(** 2019-03-25 **)
PROGRAM _INIT

	(* Always Change If Project Change *)

	//Pass Address To Global Address For External Use
	//Action, State & Status
	p_USSMEMA2Stat		:= ADR(eStat);
	p_USSMEMA2Status		:= ADR(eStatus);
	p_USSMEMA2StatTxt	:= ADR(sStatTxt);

	//Alarm
	p_USSMEMA2AlmData	:= ADR(tyAlmData);

	//Output
	p_USSMEMA2USRdy			:= ADR(bUSRdy);
	p_USSMEMA2USGdBrdRdy	:= ADR(bUSGdBrdRdy);
	p_USSMEMA2DSRdy			:= ADR(bDSRdy);
	p_USSMEMA2Transporting	:= ADR(bTransporting);
	p_USSMEMA2ConvStart		:= ADR(bConvStart);
	p_USSMEMA2ConvStop		:= ADR(bConvStop);
	p_USSMEMA2USB			:= ADR(bUSB);
	p_USSMEMA2Timer			:= ADR(bTimer);
	p_USSMEMA2Virtual		:= ADR(bVirtual);

	(* Always Change If Project Change *)

END_PROGRAM
```

#### Act_InitGlobal.st - Change By Project
```iecst
(** 2019-04-09 **)
ACTION Act_InitGlobal:

	(* Always Change If Project Change *)

	//Pass Data To Link
	p_bLinkOpsRun ACCESS p_OpsRun;

	p_eLinkConvDir ACCESS p_NtParamProjConvDir;
	p_bLinkNtParamUSWidthChkPrep ACCESS p_NtParamUSWidthChkPrep;
	p_bLinkMcParamUSWidthChkEn ACCESS p_McParamUSWidthChkEn;
	p_bLinkDIUSWidthChkSen ACCESS p_DIUSWidthChkSen;
	p_usiLinkMcMod ACCESS p_ProdRcpCurrRcp0McMod;

	//Pass Data To Internal Use
	p_udiRstErr ACCESS p_RstErrReset;
	p_bManual ACCESS p_UIMnlMod;
	p_tyParam ACCESS p_McParamUSSMEMA2Param;
	p_diTransferInTO ACCESS p_McParamTranInErrDlyTm;
	p_bLeftSen ACCESS p_DIConvLftSen;
	p_bRightSen ACCESS p_DIConvRgtSen;
	p_bUBA ACCESS p_DIUBA2;
	p_bUBAStat ACCESS p_DIUBAStat2;
	p_bVirtualEn ACCESS p_UIVSMEMAUS2En;
	p_bUBAVirtual ACCESS p_UIVSMEMAUBA2;
	p_bUBAStatVirtual ACCESS p_UIVSMEMAUBAStat2;
	p_tRstDlyTm ACCESS p_NtParamUSSMEMA2RstDlyTm;
	p_tSigInChkTm ACCESS p_NtParamUSSMEMA2SigInChkTm;
	p_sProgNm ACCESS p_NtParamUSSMEMA2ProgNm;
	p_bNtSettingsLoadDone ACCESS p_StartupNtSettingsLoadDone;

	(* Always Change If Project Change *)

END_ACTION
```

#### InputRef_Link.var - Change By Project
```iecst
(*2019-04-09*)
(**)
VAR
	p_bLinkOpsRun : REFERENCE TO BOOL;
END_VAR
(**)
VAR
	p_eLinkConvDir : REFERENCE TO eConvDir;
	p_bLinkNtParamUSWidthChkPrep : REFERENCE TO BOOL;
	p_bLinkMcParamUSWidthChkEn : REFERENCE TO BOOL;
	p_bLinkDIUSWidthChkSen : REFERENCE TO BOOL;
	p_usiLinkMcMod : REFERENCE TO USINT;
END_VAR
```

#### Act_LinkAction.st - Change By Project
```iecst
(** 2019-04-09 **)
ACTION Act_LinkAction:

	IF p_bLinkOpsRun = TRUE THEN
		p_eAct ACCESS p_OpsInvertUSSMEMA2Act;
	ELSIF p_bManual = TRUE THEN
		p_eAct ACCESS p_UIUSSMEMA2Act;
	ELSE
		p_eAct ACCESS ADR(eAct);
	END_IF

END_ACTION
```

#### Act_Link.st - Change By Project
```iecst
(** 2019-03-29 **)
ACTION Act_Link:

	//Ready Receive
	IF p_bLinkNtParamUSWidthChkPrep AND p_bLinkMcParamUSWidthChkEn THEN
		p_bRdyRcv	:= p_bLinkDIUSWidthChkSen;
	ELSE
		p_bRdyRcv	:= TRUE;
	END_IF

	//Receive Complete Signal
	//p_bComplSigOn	:= p_bLeftSen = FALSE;

	IF EDGENEG(p_bRightSen) THEN
		p_bComplSigOn	:= TRUE;
	END_IF

	IF eStat <> SMEMAActRun THEN
		p_bComplSigOn	:= FALSE;
	END_IF

	//Direction
	//	p_bDirLToR	:= p_eLinkConvDir = ConvDirLToR OR p_eLinkConvDir = ConvDirLToL;

		p_bDirLToR	:= p_eLinkConvDir = ConvDirRToL OR p_eLinkConvDir = ConvDirRToR;

END_ACTION
```

#### Cyclic.st - Do Not Change!!!
```iecst
(** 2019-03-29 **)
PROGRAM _CYCLIC

	IF bInitDone = FALSE THEN
		bInitDone	:= TRUE;

		Act_InitLocal;
		Act_InitGlobal;

	ELSIF bInitialDone = FALSE THEN
		IF p_bNtSettingsLoadDone = TRUE THEN
			bInitialDone	:= TRUE;

			Act_Initial;
		END_IF

	ELSE

		Act_RstErr;
		Act_LinkAction;
		Act_Action;
		Act_LinkEn;

		IF (p_bPrep = TRUE) AND (p_bEn = TRUE) AND (p_bDis = FALSE) THEN
			Act_Link;
			Act_Background;
			Act_Main;
		ELSE
			IF eStat <> SMEMAActIdle THEN
				eStatus	:= Done;
			ELSE
				eStatus	:= Idle;
			END_IF
		END_IF

		Act_Alarm;

	END_IF

END_PROGRAM
```

#### Act_RstErr.st - Do Not Change!!!
```iecst
(** 2018-12-08 **)
ACTION Act_RstErr:

	IF p_udiRstErr <> udiRstErrOld THEN
		bRstErr			:= TRUE;
		udiRstErrOld	:= p_udiRstErr;
	ELSE
		bRstErr			:= FALSE;
	END_IF

END_ACTION
```

#### Act_Action.st - Do Not Change!!!
```iecst
(** 2019-03-25 **)
ACTION Act_Action:

	//Reset Error
	IF (eStatus = Error) AND bRstErr THEN
		p_eAct	:= SMEMAActIdle;
		eStat	:= SMEMAActIdle;
	END_IF

	//Set p_eAct
	IF eStatus = Idle OR eStatus = Busy OR eStatus = Done THEN
		eStat	:= p_eAct;
	END_IF

END_ACTION
```

#### Act_Main.st - Do Not Change!!!
```iecst
(** 2019-03-22 **)
ACTION Act_Main:

	IF eStatOld <> eStat THEN
		fbSMEMA_Std(bEn := FALSE);
		fbSMEMA_9851(bEn := FALSE);

		bTransporting	:= FALSE;
		bConvStart		:= FALSE;
		bConvStop		:= FALSE;
		bDSRdy			:= FALSE;

		IF eStatOld <> SMEMAActIdle
			AND eStatOld <> SMEMAActSetSig
			AND eStatOld <> SMEMAActSetStatSig
			AND eStatOld <> SMEMAActRstSig
			AND eStatOld <> SMEMAActRstStatSig
			AND eStatOld <> SMEMAActSetAllSig
			AND eStatOld <> SMEMAActRstAllSig THEN

			bUSB	:= FALSE;

		END_IF

		sStatTxt	:= a_sStatText[eStat];

		eStatOld	:= eStat;

		eStatus		:= Busy;
	END_IF

	//Main
	CASE eStat OF

		SMEMAActIdle:
			IF EDGENEG(p_bManual) THEN
				bUSB	:= FALSE;
			END_IF

			eStatus	:= Idle;

		SMEMAActRun:
			IF eStatus = Idle OR eStatus = Busy THEN

				eStatus	:= Busy;

				IF p_tyParam.eSelection <> SMEMASelStandard THEN

					fbSMEMA_9851.bUSRdy			:= fbSigInChk.bSigInValid;
					fbSMEMA_9851.bRdyRcv		:= p_bRdyRcv;
					fbSMEMA_9851.bComplSigOn	:= p_bComplSigOn;

					IF p_bDirLToR = TRUE THEN

						fbSMEMA_9851.bInletSen		:= p_bLeftSen;
						fbSMEMA_9851.bOutletSen		:= p_bRightSen;

					ELSE

						fbSMEMA_9851.bInletSen		:= p_bRightSen;
						fbSMEMA_9851.bOutletSen		:= p_bLeftSen;

					END_IF

					fbSMEMA_9851.tTimeOut	:= DINT_TO_TIME(p_diTransferInTO);
					fbSMEMA_9851(bEn := TRUE);

					bTransporting	:= fbSMEMA_9851.bTransporting;
					bConvStart		:= fbSMEMA_9851.bConvStart;
					bConvStop		:= fbSMEMA_9851.bConvStop;
					bUSB			:= fbSMEMA_9851.bSigToUS AND (bTimer = FALSE) AND (bVirtual = FALSE);
					bDSRdy			:= fbSMEMA_9851.bSigToUS;

					IF fbSMEMA_9851.udiStatus = 0 THEN
						eStatus	:= Done;
					ELSIF fbSMEMA_9851.udiStatus < 65534 THEN
						eStatus		:= Error;

						IF fbSMEMA_9851.udiStatus = 1200 THEN
							udiStatus	:= 10000;	//SMEMA 9851 Transport Time Out While Transporting
						ELSIF fbSMEMA_9851.udiStatus = 1201 THEN
							udiStatus	:= 10001;	//SMEMA 9851 Transport Time Out After Opposite Machine Transport Finished
						ELSIF fbSMEMA_9851.udiStatus = 1202 THEN
							udiStatus	:= 10002;	//SMEMA 9851 Transport Time Out After Current Machine Transport Finished
						ELSIF fbSMEMA_9851.udiStatus = 1203 THEN
							udiStatus	:= 10003;	//SMEMA 9851 Transport Time Out After Both Machine Transport Finished And Waiting Outlet Sensor
						ELSE
							udiStatus	:= fbSMEMA_9851.udiStatus;
						END_IF
					END_IF

				ELSE

					fbSMEMA_Std.bUSRdy		:= fbSigInChk.bSigInValid;
					fbSMEMA_Std.bRdyRcv		:= p_bRdyRcv;
					fbSMEMA_Std.bComplSigOn	:= p_bComplSigOn;

					IF p_bDirLToR = TRUE THEN

						fbSMEMA_Std.bInletSen	:= p_bLeftSen;
						fbSMEMA_Std.bOutletSen	:= p_bRightSen;

					ELSE

						fbSMEMA_Std.bInletSen	:= p_bRightSen;
						fbSMEMA_Std.bOutletSen	:= p_bLeftSen;

					END_IF

					fbSMEMA_Std.tTimeOut	:= DINT_TO_TIME(p_diTransferInTO);
					fbSMEMA_Std(bEn := TRUE);

					bTransporting	:= fbSMEMA_Std.bTransporting;
					bConvStart		:= fbSMEMA_Std.bConvStart;
					bConvStop		:= fbSMEMA_Std.bConvStop;
					bUSB			:= fbSMEMA_Std.bSigToUS AND (bTimer = FALSE) AND (bVirtual = FALSE);
					bDSRdy			:= fbSMEMA_Std.bSigToUS;

					IF fbSMEMA_Std.udiStatus = 0 THEN
						eStatus	:= Done;
					ELSIF fbSMEMA_Std.udiStatus < 65534 THEN
						eStatus		:= Error;

						IF fbSMEMA_Std.udiStatus = 1200 THEN
							udiStatus	:= 10004;	//Standard SMEMA Transport Time Out While Transporting
						ELSIF fbSMEMA_Std.udiStatus = 1201 THEN
							udiStatus	:= 10005;	//Standard SMEMA Transport Time Out After Opposite Machine Transport Finished
						ELSIF fbSMEMA_Std.udiStatus = 1202 THEN
							udiStatus	:= 10006;	//Standard SMEMA Transport Time Out After Current Machine Transport Finished
						ELSIF fbSMEMA_Std.udiStatus = 1203 THEN
							udiStatus	:= 10007;	//Standard SMEMA Transport Time Out After Both Machine Transport Finished And Waiting Outlet Sensor
						ELSE
							udiStatus	:= fbSMEMA_Std.udiStatus;
						END_IF
					END_IF

				END_IF

			END_IF

		SMEMAActSetSig:
			IF eStatus = Idle OR eStatus = Busy THEN

				//Reset
				fbSMEMA_Std(bEn := FALSE);
				fbSMEMA_9851(bEn := FALSE);

				bConvStart	:= FALSE;
				bConvStop	:= FALSE;

				bUSB	:= TRUE;
				eStatus	:= Done;

			END_IF

		SMEMAActSetStatSig:
			IF eStatus = Idle OR eStatus = Busy THEN

				//Reset
				fbSMEMA_Std(bEn := FALSE);
				fbSMEMA_9851(bEn := FALSE);

				bConvStart	:= FALSE;
				bConvStop	:= FALSE;

				eStatus	:= Done;

			END_IF

		SMEMAActRstSig:
			IF eStatus = Idle OR eStatus = Busy THEN

				//Reset
				fbSMEMA_Std(bEn := FALSE);
				fbSMEMA_9851(bEn := FALSE);

				bConvStart	:= FALSE;
				bConvStop	:= FALSE;

				bUSB	:= FALSE;
				eStatus	:= Done;

			END_IF

		SMEMAActRstStatSig:
			IF eStatus = Idle OR eStatus = Busy THEN

				//Reset
				fbSMEMA_Std(bEn := FALSE);
				fbSMEMA_9851(bEn := FALSE);

				bConvStart	:= FALSE;
				bConvStop	:= FALSE;

				eStatus	:= Done;

			END_IF

		SMEMAActSetAllSig:
			IF eStatus = Idle OR eStatus = Busy THEN

				//Reset
				fbSMEMA_Std(bEn := FALSE);
				fbSMEMA_9851(bEn := FALSE);

				bConvStart	:= FALSE;
				bConvStop	:= FALSE;

				bUSB	:= TRUE;
				eStatus	:= Done;

			END_IF

		SMEMAActRstAllSig:
			IF eStatus = Idle OR eStatus = Busy THEN

				//Reset
				fbSMEMA_Std(bEn := FALSE);
				fbSMEMA_9851(bEn := FALSE);

				bConvStart	:= FALSE;
				bConvStop	:= FALSE;

				bUSB	:= FALSE;
				eStatus	:= Done;

			END_IF

	END_CASE

END_ACTION
```

#### Act_Alarm.st - Do Not Change!!!
```iecst
(** 2019-03-25 **)
ACTION Act_Alarm:

	//Error
	IF EDGEPOS(eStatus = Error) THEN

		tyAlmData.sProgNm		:= p_sProgNm;
		tyAlmData.udiCode		:= udiStatus;
		tyAlmData.eSeverity		:= AlmSeverityError;
		tyAlmData.udiRunTime	:= tyAlmData.udiRunTime + 1;
		tyAlmData.bAlm			:= TRUE;
		tyAlmData.udiModuleNum  := udiModuleNum;
		g_sUSSMEMAProgNm		:= p_sProgNm;

		//Get Error Message
		IF tyAlmData.udiCode < 10000 OR tyAlmData.udiCode > 10099 THEN
			tyAlmData.sAlmMsg	:= 'Unknown';
			tyAlmData.sRcyMsg	:= 'Unknown';
		ELSE
			tyAlmData.sAlmMsg	:= a_tyAlmText[tyAlmData.udiCode].sAlmText;
			tyAlmData.sRcyMsg	:= a_tyAlmText[tyAlmData.udiCode].sRcyText;
		END_IF

		sStatTxt	:= tyAlmData.sAlmMsg;

	ELSIF bRstErr AND (tyAlmData.udiCode <> 0) THEN

		tyAlmData.udiCode	:= 0;
		tyAlmData.eSeverity	:= AlmSeverityNA;
		tyAlmData.sAlmMsg	:= '';
		tyAlmData.sRcyMsg	:= '';
		tyAlmData.bAlm			:= FALSE;

		sStatTxt	:= a_sStatText[eStat];

	END_IF

END_ACTION
```

#### Local.var - Do Not Change!!!
```iecst
(*2019-04-30*)
(**)
(*Local Action, State & Status*)
VAR
	eAct : eSMEMAAction := SMEMAActIdle;
	eStat : eSMEMAAction := SMEMAActIdle;
	eStatus : eFBStatus := Idle;
	udiStatus : UDINT := 0;
	sStatTxt : STRING[200] := '';
	a_sStatText : ARRAY[0..50] OF STRING[200] := ['Idling','Upstream SMEMA Running','Turning On USB Signal','NA','Turning Off USB Signal','NA','Turning On USB Signal','Turning Off USB Signal',43('')];
END_VAR
(**)
(*Local Alarm*)
VAR
	tyAlmData : tyAlmDat;
	a_tyAlmText : ARRAY[10000..10099] OF tyAlmTxt := [(sAlmText:='SMEMA 9851 Transport Time Out While Transporting',sRcyText:='Timeout Expired Before Operation Completed. Reset And Resume Operation.'),(sAlmText:='SMEMA 9851 Transport Time Out After Opposite Machine Transport Finished',sRcyText:='Timeout Expired Before Operation Completed. Reset And Resume Operation.'),(sAlmText:='SMEMA 9851 Transport Time Out After Current Machine Transport Finished',sRcyText:='Timeout Expired Before Operation Completed. Reset And Resume Operation.'),(sAlmText:='SMEMA 9851 Transport Time Out After Both Machine Transport Finished And Waiting Outlet Sensor',sRcyText:='Timeout Expired Before Operation Completed. Reset And Resume Operation.'),(sAlmText:='Standard SMEMA Transport Time Out While Transporting',sRcyText:='Timeout Expired Before Operation Completed. Reset And Resume Operation.'),(sAlmText:='Standard SMEMA Transport Time Out After Opposite Machine Transport Finished',sRcyText:='Timeout Expired Before Operation Completed. Reset And Resume Operation.'),(sAlmText:='Standard SMEMA Transport Time Out After Current Machine Transport Finished',sRcyText:='Timeout Expired Before Operation Completed. Reset And Resume Operation.'),(sAlmText:='Standard SMEMA Transport Time Out After Both Machine Transport Finished And Waiting Outlet Sensor',sRcyText:='Timeout Expired Before Operation Completed. Reset And Resume Operation.'),92((0))];
END_VAR
(**)
(*Local Output*)
VAR
	bUSRdy : BOOL := FALSE;
	bUSGdBrdRdy : BOOL := FALSE;
	bDSRdy : BOOL := FALSE;
	bTransporting : BOOL := FALSE;
	bConvStart : BOOL := FALSE;
	bConvStop : BOOL := FALSE;
	bUSB : BOOL := FALSE;
	bTimer : BOOL;
	bVirtual : BOOL;
END_VAR
(**)
(*Local Input*)
VAR
	udiRstErr : UDINT := 0;
	bPrep : BOOL := TRUE;
	bEn : BOOL := TRUE;
	bDis : BOOL := FALSE;
	bManual : BOOL := FALSE;
	tyParam : tySMEMAParam;
	diTransferInTO : DINT := 20000;
	bDirLToR : BOOL := FALSE;
	bRdyRcv : BOOL := TRUE;
	bLeftSen : BOOL := FALSE;
	bRightSen : BOOL := FALSE;
	bComplSigOn : BOOL := FALSE;
	bUBA : BOOL := FALSE;
	bUBAStat : BOOL := FALSE;
	bTimerEnSen : BOOL;
	bTimerEnSenEdge : BOOL;
	bVirtualEn : BOOL;
	bUBAVirtual : BOOL;
	bUBAStatVirtual : BOOL;
	tRstDlyTm : TIME := T#500ms;
	tSigInChkTm : TIME := T#100ms;
	sProgNm : STRING[15] := 'USSMEMA2';
	bNtSettingsLoadDone : BOOL := TRUE;
END_VAR
(**)
(*Local*)
VAR
	bRstErr : BOOL;
	udiRstErrOld : UDINT;
	bInitDone : BOOL;
	bInitialDone : BOOL;
	fbTimerDlyTm : TON := (PT:=T#1s);
	fbTimeTrig : R_TRIG;
	fbSMEMA_Std : fbSMEMAUS_Std;
	fbSMEMA_9851 : fbSMEMAUS_9851;
	fbSigInChk : fbSMEMASigInChk;
	eStatOld : eSMEMAAction := SMEMAActIdle;
	udiModuleNum : UDINT := 2701;
END_VAR
```

### Pneu.typ - Do Not Change!!!
```iecst
(*2018-12-11*)
(**)
(*Action*)

TYPE
	ePneuAction :
		(
		PneuActIdle,
		PneuActSetAll,
		PneuActRstAll,
		PneuActSetExt,
		PneuActSetRet,
		PneuActExt,
		PneuActRet,
		PneuActExtSenToMidSen,
		PneuActMidSenToRetSen,
		PneuActRetSenToMidSen,
		PneuActMidSenToExtSen
		);
END_TYPE

(**)

TYPE
	eClampType :
		(
		ClampNoRS := 0,
		ThreeClampsWithRS := 1
		);
END_TYPE
```

### PneuNoSenStopper.var - Change By Project
```iecst
(*2019-03-25*)
(**)
(*Action & State & Status*)
VAR
	p_PneuNoSenStopperStat : UDINT;
	p_PneuNoSenStopperStatus : UDINT;
	p_PneuNoSenStopperStatTxt : UDINT;
END_VAR
(**)
(*Alarm*)
VAR
	p_PneuNoSenStopperAlmData : UDINT;
END_VAR
(**)
(*Output*)
VAR
	p_PneuNoSenStopperExtCtrl : UDINT;
	p_PneuNoSenStopperRetCtrl : UDINT;
	p_PneuNoSenStopperTwoCtrlOut : UDINT;
	p_PneuNoSenStopperExtended : UDINT;
	p_PneuNoSenStopperRetracted : UDINT;
END_VAR
```

### Program Logical/Pneu/PneuNoSenStopper (IEC, version 1.00.0) - 1.00.0 - NtPneu v5.00.0

#### Init.st - Change By Project
```iecst
(** 2019-03-25 **)
PROGRAM _INIT

	(* Always Change If Project Change *)

	//Pass Address To Global Address For External Use
	//Action, State & Status
	p_PneuNoSenStopperStat			:= ADR(eStat);
	p_PneuNoSenStopperStatus		:= ADR(eStatus);
	p_PneuNoSenStopperStatTxt		:= ADR(sStatTxt);

	//Alarm
	p_PneuNoSenStopperAlmData		:= ADR(tyAlmData);

	//Output
	p_PneuNoSenStopperExtCtrl		:= ADR(bExtCtrl);
	p_PneuNoSenStopperRetCtrl		:= ADR(bRetCtrl);
	p_PneuNoSenStopperTwoCtrlOut	:= ADR(bTwoCtrlOut);
	p_PneuNoSenStopperExtended		:= ADR(bExtended);
	p_PneuNoSenStopperRetracted		:= ADR(bRetracted);

	(* Always Change If Project Change *)

END_PROGRAM
```

#### Act_InitGlobal.st - Change By Project
```iecst
(** 2019-04-09 **)
ACTION Act_InitGlobal:

	(* Always Change If Project Change *)

	//Pass Data To Link
	p_bLinkOpsRun ACCESS p_OpsRun;
	p_bLinkOpsSimu ACCESS p_SimuRun;

	p_bLinkDISafetyRlySig ACCESS p_DISafetyRlySig;

	//Pass Data To Internal Use
	p_udiRstErr ACCESS p_RstErrReset;
	p_bPrep ACCESS p_NtParamProjStopperPrep;
	p_bDis ACCESS p_McParamStopperDis;
	p_bManual ACCESS p_UIMnlMod;
	p_bTwoCtrlIn ACCESS p_NtParamStopperTwoCtrlIn;
	p_sProgNm ACCESS p_NtParamStopperProgNm;
	p_tExtDlyTm ACCESS p_NtParamStopperExtDlyTm;
	p_tRetDlyTm ACCESS p_NtParamStopperRetDlyTm;
	p_bNtSettingsLoadDone ACCESS p_StartupNtSettingsLoadDone;

	(* Always Change If Project Change *)

END_ACTION
```

#### Act_LinkAction.st - Change By Project
```iecst
(** 2019-04-09 **)
ACTION Act_LinkAction:

	IF p_bLinkOpsRun = TRUE THEN
		p_eAct ACCESS p_OpsInvertStopperAct;
	ELSIF p_bLinkOpsSimu = TRUE THEN
		p_eAct ACCESS p_SimuInvStopperAct;
	ELSIF p_bManual = TRUE THEN
		p_eAct ACCESS p_UIStopperAct;
	ELSE
		p_eAct ACCESS ADR(eAct);
	END_IF

END_ACTION
```

#### Act_InitLocal.st - Do Not Change!!!
```iecst
(** 2019-03-25 **)
ACTION Act_InitLocal:

	//Input Reference Link To Local Variable
	p_eAct ACCESS ADR(eAct);
	p_udiRstErr ACCESS ADR(udiRstErr);
	p_bPrep ACCESS ADR(bPrep);
	p_bEn ACCESS ADR(bEn);
	p_bDis ACCESS ADR(bDis);
	p_bManual ACCESS ADR(bManual);
	p_bTwoCtrlIn ACCESS ADR(bTwoCtrlIn);
	p_bExtSafetySen ACCESS ADR(bExtSafetySen);
	p_bRetSafetySen ACCESS ADR(bRetSafetySen);
	p_sProgNm ACCESS ADR(sProgNm);
	p_tExtDlyTm ACCESS ADR(tExtDlyTm);
	p_tRetDlyTm ACCESS ADR(tRetDlyTm);
	p_bNtSettingsLoadDone ACCESS ADR(bNtSettingsLoadDone);

END_ACTION
```

#### Act_Initial.st - Do Not Change!!!
```iecst
(** 2019-03-22 **)
ACTION Act_Initial:

	//Initial
	sStatTxt	:= a_sStatText[eStat];

	bTwoCtrlOut	:= p_bTwoCtrlIn;

	fbPneuExtChk.tDlyTm	:= p_tExtDlyTm;
	fbPneuExtChk(bEn := FALSE);

	fbPneuRetChk.tDlyTm	:= p_tRetDlyTm;
	fbPneuRetChk(bEn := FALSE);

END_ACTION
```

#### Act_Alarm.st - Do Not Change!!!
```iecst
(** 2019-03-25 **)
ACTION Act_Alarm:

	//Error
	IF EDGEPOS(eStatus = Error) THEN

		tyAlmData.sProgNm		:= p_sProgNm;
		tyAlmData.udiCode		:= udiStatus;
		tyAlmData.eSeverity		:= AlmSeverityError;
		tyAlmData.udiRunTime	:= tyAlmData.udiRunTime + 1;
		tyAlmData.bAlm			:= TRUE;
		tyAlmData.udiModuleNum  := udiModuleNum;
		g_sPneuNoSenProgNm		:= p_sProgNm;

		//Get Error Message
		IF tyAlmData.udiCode < 10000 OR tyAlmData.udiCode > 10099 THEN
			tyAlmData.sAlmMsg	:= 'Unknown';
			tyAlmData.sRcyMsg	:= 'Unknown';
		ELSE
			tyAlmData.sAlmMsg	:= a_tyAlmText[tyAlmData.udiCode].sAlmText;
			tyAlmData.sRcyMsg	:= a_tyAlmText[tyAlmData.udiCode].sRcyText;
		END_IF

		sStatTxt	:= tyAlmData.sAlmMsg;

	ELSIF bRstErr AND (tyAlmData.udiCode <> 0) THEN

		tyAlmData.udiCode	:= 0;
		tyAlmData.eSeverity	:= AlmSeverityNA;
		tyAlmData.sAlmMsg	:= '';
		tyAlmData.sRcyMsg	:= '';
		tyAlmData.bAlm		:= FALSE;
		sStatTxt	:= a_sStatText[eStat];

	END_IF

END_ACTION
```

#### InputRef.var - Do Not Change!!!
```iecst
(*2019-03-25*)
(**)
(*General*)
VAR
	p_eAct : REFERENCE TO ePneuAction;
	p_udiRstErr : REFERENCE TO UDINT;
	p_bPrep : REFERENCE TO BOOL;
	p_bEn : REFERENCE TO BOOL;
	p_bDis : REFERENCE TO BOOL;
END_VAR
(**)
(*Configuration*)
VAR
	p_bManual : REFERENCE TO BOOL;
	p_bTwoCtrlIn : REFERENCE TO BOOL;
	p_bExtSafetySen : REFERENCE TO BOOL;
	p_bRetSafetySen : REFERENCE TO BOOL;
	p_sProgNm : REFERENCE TO STRING[15];
	p_tExtDlyTm : REFERENCE TO TIME;
	p_tRetDlyTm : REFERENCE TO TIME;
	p_bNtSettingsLoadDone : REFERENCE TO BOOL;
END_VAR
```

#### Local.var - Do Not Change!!!
```iecst
(*2019-04-30*)
(**)
(*Local Action, State & Status*)
VAR
	eAct : ePneuAction := PneuActIdle;
	eStat : ePneuAction := PneuActIdle;
	eStatus : eFBStatus := Idle;
	udiStatus : UDINT := 0;
	sStatTxt : STRING[200] := '';
	a_sStatText : ARRAY[0..50] OF STRING[200] := ['Idling','Set All','Reset All','Set Extend','Set Retract','Extending','Retracting','Retracting From Extend Sensor To Middle Sensor','Retracting From Middle Sensor To Retract Sensor','Extending From Retract Sensor To Middle Sensor','Extending From Middle Sensor To Extend Sensor',40('')];
END_VAR
(**)
(*Local Alarm*)
VAR
	tyAlmData : tyAlmDat;
	a_tyAlmText : ARRAY[10000..10099] OF tyAlmTxt := [(sAlmText:='Safety Check Error While Extending',sRcyText:='Safety System Has Been Triggered. All Operations Are Disable. Remove the Obstacle That Triggered The Safety Interlock To Resume Operation.'),(sAlmText:='Extend Sensor On Checking Time Out While Extending',sRcyText:='Sensor Timeout Expired Before Operation Completed. Sensor Operation Is Abnormal. Solve The Error To Resume Operation. '),(sAlmText:='Retract Sensor Off Checking Time Out While Extending',sRcyText:='Sensor Timeout Expired Before Operation Completed. Sensor Operation Is Abnormal. Solve The Error To Resume Operation.'),(sAlmText:='Safety Check Error While Retracting',sRcyText:='Safety System Has Been Triggered. All Operations Are Disable. Remove the Obstacle That Triggered The Safety Interlock To Resume Operation.'),(sAlmText:='Retract Sensor On Checking Time Out While Retracting',sRcyText:='Sensor Timeout Expired Before Operation Completed. Sensor Operation Is Abnormal. Solve The Error To Resume Operation.'),(sAlmText:='Extend Sensor Off Checking Time Out While Retracting',sRcyText:='Sensor Timeout Expired Before Operation Completed. Sensor Operation Is Abnormal. Solve The Error To Resume Operation.'),94((0))];
END_VAR
(**)
(*Local Output*)
VAR
	bExtCtrl : BOOL;
	bRetCtrl : BOOL;
	bTwoCtrlOut : BOOL := FALSE;
	bExtended : BOOL := FALSE;
	bRetracted : BOOL := FALSE;
END_VAR
(**)
(*Local Input*)
VAR
	udiRstErr : UDINT := 0;
	bPrep : BOOL := TRUE;
	bEn : BOOL := TRUE;
	bDis : BOOL := FALSE;
	bManual : BOOL := FALSE;
	bTwoCtrlIn : BOOL := FALSE;
	bExtSafetySen : BOOL := TRUE;
	bRetSafetySen : BOOL := TRUE;
	sProgNm : STRING[15] := 'PneuNoSen';
	tExtDlyTm : TIME := T#1s;
	tRetDlyTm : TIME := T#1s;
	bNtSettingsLoadDone : BOOL := TRUE;
END_VAR
(**)
(*Local*)
VAR
	bRstErr : BOOL;
	udiRstErrOld : UDINT;
	bInitDone : BOOL;
	bInitialDone : BOOL;
	fbPneuExtChk : fbPneuNoSenExtChk;
	fbPneuRetChk : fbPneuNoSenRetChk;
	eStatOld : ePneuAction := PneuActIdle;
	udiModuleNum : UDINT := 2401;
END_VAR
```

### PneuNoSenClamp.var - Change By Project
```iecst
(*2019-03-25*)
(**)
(*Action & State & Status*)
VAR
	p_PneuNoSenClampStat : UDINT;
	p_PneuNoSenClampStatus : UDINT;
	p_PneuNoSenClampStatTxt : UDINT;
END_VAR
(**)
(*Alarm*)
VAR
	p_PneuNoSenClampAlmData : UDINT;
END_VAR
(**)
(*Output*)
VAR
	p_PneuNoSenClampExtCtrl : UDINT;
	p_PneuNoSenClampRetCtrl : UDINT;
	p_PneuNoSenClampTwoCtrlOut : UDINT;
	p_PneuNoSenClampExtended : UDINT;
	p_PneuNoSenClampRetracted : UDINT;
END_VAR
```

### Program Logical/Pneu/PneuNoSenClamp (IEC) - 1.00.0 - NtPneu v5.00.0

#### InputRef.var
```iecst
(*2020-10-08*)
(**)
(*General*)
VAR
	p_eAct : REFERENCE TO ePneuAction;
	p_udiRstErr : REFERENCE TO UDINT;
	p_bPrep : REFERENCE TO BOOL;
	p_bEn : REFERENCE TO BOOL;
	p_bDis : REFERENCE TO BOOL;
END_VAR
(**)
(*Configuration*)
VAR
	p_bClampPrep : REFERENCE TO BOOL;
	p_eClampOption : REFERENCE TO eClampType;
	p_bManual : REFERENCE TO BOOL;
	p_bTwoCtrlIn : REFERENCE TO BOOL;
	p_bExtSafetySen : REFERENCE TO BOOL;
	p_bRetSafetySen : REFERENCE TO BOOL;
	p_sProgNm : REFERENCE TO STRING[15];
	p_tExtDlyTm : REFERENCE TO TIME;
	p_tRetDlyTm : REFERENCE TO TIME;
	p_bNtSettingsLoadDone : REFERENCE TO BOOL;
END_VAR
```

#### InputRef_Link.var
```iecst
(*2019-04-09*)
(**)
(*External*)
VAR
	p_bLinkOpsRun : REFERENCE TO BOOL;
END_VAR
(**)
VAR
	p_bLinkDISafetyRlySig : REFERENCE TO BOOL;
END_VAR
```

#### Local.var
```iecst
(*2020-10-08*)
(**)
(*Local Action, State & Status*)
VAR
	eAct : ePneuAction := PneuActIdle;
	eStat : ePneuAction := PneuActIdle;
	eStatus : eFBStatus := Idle;
	udiStatus : UDINT := 0;
	sStatTxt : STRING[200] := '';
	a_sStatText : ARRAY[0..50] OF STRING[200] := ['Idling','Set All','Reset All','Set Extend','Set Retract','Extending','Retracting','Retracting From Extend Sensor To Middle Sensor','Retracting From Middle Sensor To Retract Sensor','Extending From Retract Sensor To Middle Sensor','Extending From Middle Sensor To Extend Sensor',40('')];
END_VAR
(**)
(*Local Alarm*)
VAR
	tyAlmData : tyAlmDat;
	a_tyAlmText : ARRAY[10000..10099] OF tyAlmTxt := [(sAlmText:='Safety Check Error While Extending',sRcyText:='Safety System Has Been Triggered. All Operations Are Disable. Remove the Obstacle That Triggered The Safety Interlock To Resume Operation.'),(sAlmText:='Extend Sensor On Checking Time Out While Extending',sRcyText:='Sensor Timeout Expired Before Operation Completed. Sensor Operation Is Abnormal. Solve The Error To Resume Operation. '),(sAlmText:='Retract Sensor Off Checking Time Out While Extending',sRcyText:='Sensor Timeout Expired Before Operation Completed. Sensor Operation Is Abnormal. Solve The Error To Resume Operation.'),(sAlmText:='Safety Check Error While Retracting',sRcyText:='Safety System Has Been Triggered. All Operations Are Disable. Remove the Obstacle That Triggered The Safety Interlock To Resume Operation.'),(sAlmText:='Retract Sensor On Checking Time Out While Retracting',sRcyText:='Sensor Timeout Expired Before Operation Completed. Sensor Operation Is Abnormal. Solve The Error To Resume Operation.'),(sAlmText:='Extend Sensor Off Checking Time Out While Retracting',sRcyText:='Sensor Timeout Expired Before Operation Completed. Sensor Operation Is Abnormal. Solve The Error To Resume Operation.'),94((0))];
END_VAR
(**)
(*Local Output*)
VAR
	bExtCtrl : BOOL;
	bRetCtrl : BOOL;
	bTwoCtrlOut : BOOL := FALSE;
	bExtended : BOOL := FALSE;
	bRetracted : BOOL := FALSE;
END_VAR
(**)
(*Local Input*)
VAR
	udiRstErr : UDINT := 0;
	bPrep : BOOL := TRUE;
	bEn : BOOL := TRUE;
	bDis : BOOL := FALSE;
	bClampPrep : BOOL := FALSE;
	eClampOption : eClampType := ClampNoRS;
	bManual : BOOL := FALSE;
	bTwoCtrlIn : BOOL := FALSE;
	bExtSafetySen : BOOL := TRUE;
	bRetSafetySen : BOOL := TRUE;
	sProgNm : STRING[15] := 'PneuNoSen';
	tExtDlyTm : TIME := T#1s;
	tRetDlyTm : TIME := T#1s;
	bNtSettingsLoadDone : BOOL := TRUE;
END_VAR
(**)
(*Local*)
VAR
	bRstErr : BOOL;
	udiRstErrOld : UDINT;
	bInitDone : BOOL;
	bInitialDone : BOOL;
	fbPneuExtChk : fbPneuNoSenExtChk;
	fbPneuRetChk : fbPneuNoSenRetChk;
	eStatOld : ePneuAction := PneuActIdle;
	udiModuleNum : UDINT := 2401;
END_VAR
```

#### Act_InitGlobal.st
```iecst
(** 2020-10-08 **)
ACTION Act_InitGlobal:

	(* Always Change If Project Change *)

	//Pass Data To Link
	p_bLinkOpsRun ACCESS p_OpsRun;

	p_bLinkDISafetyRlySig ACCESS p_DISafetyRlySig;

	//Pass Data To Internal Use
	p_udiRstErr ACCESS p_RstErrReset;
	p_bDis ACCESS p_McParamClampDis;
	p_bManual ACCESS p_UIMnlMod;
	p_bTwoCtrlIn ACCESS p_NtParamClampTwoCtrlIn;
	p_sProgNm ACCESS p_NtParamClampProgNm;
	p_tExtDlyTm ACCESS p_NtParamClampExtDlyTm;
	p_tRetDlyTm ACCESS p_NtParamClampRetDlyTm;
	p_bNtSettingsLoadDone ACCESS p_StartupNtSettingsLoadDone;

	p_bClampPrep ACCESS p_NtParamProjClampPrep;
	p_eClampOption ACCESS p_NtParamProjClampOption;

	(* Always Change If Project Change *)

END_ACTION
```

#### Act_InitLocal.st
```iecst
(** 2020-10-08 **)
ACTION Act_InitLocal:

	//Input Reference Link To Local Variable
	p_eAct ACCESS ADR(eAct);
	p_udiRstErr ACCESS ADR(udiRstErr);
	p_bPrep ACCESS ADR(bPrep);
	p_bEn ACCESS ADR(bEn);
	p_bDis ACCESS ADR(bDis);
	p_bClampPrep ACCESS ADR(bClampPrep);
	p_eClampOption ACCESS ADR(eClampOption);
	p_bManual ACCESS ADR(bManual);
	p_bTwoCtrlIn ACCESS ADR(bTwoCtrlIn);
	p_bExtSafetySen ACCESS ADR(bExtSafetySen);
	p_bRetSafetySen ACCESS ADR(bRetSafetySen);
	p_sProgNm ACCESS ADR(sProgNm);
	p_tExtDlyTm ACCESS ADR(tExtDlyTm);
	p_tRetDlyTm ACCESS ADR(tRetDlyTm);
	p_bNtSettingsLoadDone ACCESS ADR(bNtSettingsLoadDone);

END_ACTION
```

#### Act_LinkAction.st
```iecst
(** 2019-04-09 **)
ACTION Act_LinkAction:

	IF p_bLinkOpsRun = TRUE THEN
		p_eAct ACCESS p_OpsInvertClampAct;
	ELSIF p_bManual = TRUE THEN
		p_eAct ACCESS p_UIClampAct;
	ELSE
		p_eAct ACCESS ADR(eAct);
	END_IF

END_ACTION
```

#### Act_LinkEn.st
```iecst
(** 2020-10-08 **)
ACTION Act_LinkEn:

	//Link bPrep, bEn & bDis
	p_bPrep := p_bClampPrep AND (p_eClampOption=ClampNoRS);
END_ACTION
```

#### Act_Main.st
```iecst
(** 2019-01-10 **)
ACTION Act_Main:

	IF eStatOld <> eStat THEN
		fbPneuExtChk(bEn := FALSE);
		fbPneuRetChk(bEn := FALSE);

		sStatTxt	:= a_sStatText[eStat];

		eStatOld	:= eStat;

		eStatus		:= Busy;
	END_IF

	//Main
	CASE eStat OF

		PneuActIdle:
			eStatus	:= Idle;

		PneuActSetAll:
			IF eStatus = Idle OR eStatus = Busy THEN

				//Reset
				fbPneuExtChk(bEn := FALSE);
				fbPneuRetChk(bEn := FALSE);

				bExtCtrl	:= TRUE;
				bRetCtrl	:= TRUE;

				bExtended	:= FALSE;
				bRetracted	:= FALSE;

				eStatus	:= Done;

			END_IF

		PneuActRstAll:
			IF eStatus = Idle OR eStatus = Busy THEN

				//Reset
				fbPneuExtChk(bEn := FALSE);
				fbPneuRetChk(bEn := FALSE);

				bExtCtrl	:= FALSE;
				bRetCtrl	:= FALSE;

				bExtended	:= FALSE;
				bRetracted	:= FALSE;

				eStatus	:= Done;

			END_IF

		PneuActSetExt:
			IF eStatus = Idle OR eStatus = Busy THEN

				//Reset
				fbPneuExtChk(bEn := FALSE);
				fbPneuRetChk(bEn := FALSE);

				bExtCtrl	:= TRUE;
				bRetCtrl	:= FALSE;

				bExtended	:= TRUE;
				bRetracted	:= FALSE;

				eStatus	:= Done;

			END_IF

		PneuActSetRet:
			IF eStatus = Idle OR eStatus = Busy THEN

				//Reset
				fbPneuExtChk(bEn := FALSE);
				fbPneuRetChk(bEn := FALSE);

				bExtCtrl	:= FALSE;
				bRetCtrl	:= TRUE;

				bExtended	:= FALSE;
				bRetracted	:= TRUE;

				eStatus	:= Done;

			END_IF

		PneuActExt:
			IF eStatus = Idle OR eStatus = Busy THEN

				eStatus	:= Busy;

				//Reset
				fbPneuRetChk(bEn := FALSE);

				bExtCtrl	:= TRUE;
				bRetCtrl	:= FALSE;

				fbPneuExtChk.bExtSafety	:= p_bExtSafetySen;
				fbPneuExtChk(bEn := TRUE);

				IF fbPneuExtChk.udiStatus = 0 THEN
					bExtended	:= TRUE;
					bRetracted	:= FALSE;
					eStatus		:= Done;
				ELSIF fbPneuExtChk.udiStatus < 65534 THEN
					IF p_bTwoCtrlIn = TRUE THEN
						bExtCtrl	:= FALSE;
						bRetCtrl	:= FALSE;
					ELSE
						bExtCtrl	:= FALSE;
						bRetCtrl	:= TRUE;
					END_IF

					bExtended	:= FALSE;
					bRetracted	:= FALSE;

					eStatus		:= Error;

					IF fbPneuExtChk.udiStatus = 1507 THEN
						udiStatus	:= 10000;	//Safety Check Error While Extending
					ELSE
						udiStatus	:= fbPneuExtChk.udiStatus;
					END_IF
				END_IF

			END_IF

		PneuActRet:
			IF eStatus = Idle OR eStatus = Busy THEN

				eStatus	:= Busy;

				//Reset
				fbPneuExtChk(bEn := FALSE);

				bExtCtrl	:= FALSE;
				bRetCtrl	:= TRUE;

				fbPneuRetChk.bRetSafety	:= p_bRetSafetySen;
				fbPneuRetChk(bEn := TRUE);

				IF fbPneuRetChk.udiStatus = 0 THEN
					bExtended	:= FALSE;
					bRetracted	:= TRUE;
					eStatus		:= Done;
				ELSIF fbPneuRetChk.udiStatus < 65534 THEN
					IF p_bTwoCtrlIn = TRUE THEN
						bExtCtrl	:= FALSE;
						bRetCtrl	:= FALSE;
					ELSE
						bExtCtrl	:= TRUE;
						bRetCtrl	:= FALSE;
					END_IF

					bExtended	:= FALSE;
					bRetracted	:= FALSE;

					eStatus		:= Error;

					IF fbPneuRetChk.udiStatus = 1508 THEN
						udiStatus	:= 10003;	//Safety Check Error While Retracting
					ELSE
						udiStatus	:= fbPneuRetChk.udiStatus;
					END_IF
				END_IF

			END_IF

		ELSE
			IF eStatus = Idle OR eStatus = Busy THEN
				eStatus	:= Done;
			END_IF

	END_CASE

END_ACTION
```

#### Act_RstErr.st
```iecst
(** 2018-12-11 **)
ACTION Act_RstErr:

	IF p_udiRstErr <> udiRstErrOld THEN
		bRstErr			:= TRUE;
		udiRstErrOld	:= p_udiRstErr;
	ELSE
		bRstErr			:= FALSE;
	END_IF

END_ACTION
```

#### Cyclic.st
```iecst
(** 2019-03-29 **)
PROGRAM _CYCLIC

	IF bInitDone = FALSE THEN
		bInitDone	:= TRUE;

		Act_InitLocal;
		Act_InitGlobal;

	ELSIF bInitialDone = FALSE THEN
		IF p_bNtSettingsLoadDone = TRUE THEN
			bInitialDone	:= TRUE;

			Act_Initial;
		END_IF

	ELSE

		Act_RstErr;
		Act_LinkAction;
		Act_Action;
		Act_LinkEn;

		IF (p_bPrep = TRUE) AND (p_bEn = TRUE) AND (p_bDis = FALSE) THEN
			Act_Link;
			Act_Main;
		ELSE
			IF eStat <> PneuActIdle THEN
				IF eStat = PneuActSetExt OR eStat = PneuActExt THEN
					bExtended	:= TRUE;
					bRetracted	:= FALSE;
				ELSIF eStat = PneuActSetRet OR eStat = PneuActRet THEN
					bExtended	:= FALSE;
					bRetracted	:= TRUE;
				END_IF

				eStatus	:= Done;
			ELSE
				eStatus	:= Idle;
			END_IF
		END_IF

		Act_Alarm;

	END_IF

END_PROGRAM
```

#### Init.st
```iecst
(** 2019-03-25 **)
PROGRAM _INIT

	(* Always Change If Project Change *)

	//Pass Address To Global Address For External Use
	//Action, State & Status
	p_PneuNoSenClampStat		:= ADR(eStat);
	p_PneuNoSenClampStatus		:= ADR(eStatus);
	p_PneuNoSenClampStatTxt		:= ADR(sStatTxt);

	//Alarm
	p_PneuNoSenClampAlmData		:= ADR(tyAlmData);

	//Output
	p_PneuNoSenClampExtCtrl		:= ADR(bExtCtrl);
	p_PneuNoSenClampRetCtrl		:= ADR(bRetCtrl);
	p_PneuNoSenClampTwoCtrlOut	:= ADR(bTwoCtrlOut);
	p_PneuNoSenClampExtended	:= ADR(bExtended);
	p_PneuNoSenClampRetracted	:= ADR(bRetracted);

	(* Always Change If Project Change *)

END_PROGRAM
```

### Pneu2SenInShutter.var - Change By Project
```iecst
(*2019-03-25*)
(**)
(*Action & State & Status*)
VAR
	p_Pneu2SenInShutterStat : UDINT;
	p_Pneu2SenInShutterStatus : UDINT;
	p_Pneu2SenInShutterStatTxt : UDINT;
END_VAR
(**)
(*Alarm*)
VAR
	p_Pneu2SenInShutterAlmData : UDINT;
END_VAR
(**)
(*Output*)
VAR
	p_Pneu2SenInShutterExtCtrl : UDINT;
	p_Pneu2SenInShutterRetCtrl : UDINT;
	p_Pneu2SenInShutterTwoCtrlOut : UDINT;
	p_Pneu2SenInShutterExtended : UDINT;
	p_Pneu2SenInShutterRetracted : UDINT;
END_VAR
```

### Program Logical/Pneu/Pneu2SenInShutter (IEC, version 1.00.0) - 1.00.0 - NtPneu v5.00.0

#### Init.st - Change By Project
```iecst
(** 2019-03-25 **)
PROGRAM _INIT

	(* Always Change If Project Change *)

	//Pass Address To Global Address For External Use
	//Action, State & Status
	p_Pneu2SenInShutterStat			:= ADR(eStat);
	p_Pneu2SenInShutterStatus		:= ADR(eStatus);
	p_Pneu2SenInShutterStatTxt		:= ADR(sStatTxt);

	//Alarm
	p_Pneu2SenInShutterAlmData		:= ADR(tyAlmData);

	//Output
	p_Pneu2SenInShutterExtCtrl		:= ADR(bExtCtrl);
	p_Pneu2SenInShutterRetCtrl		:= ADR(bRetCtrl);
	p_Pneu2SenInShutterTwoCtrlOut	:= ADR(bTwoCtrlOut);
	p_Pneu2SenInShutterExtended		:= ADR(bExtended);
	p_Pneu2SenInShutterRetracted	:= ADR(bRetracted);

	(* Always Change If Project Change *)

END_PROGRAM
```

#### Act_InitGlobal.st - Change By Project
```iecst
(** 2019-04-09 **)
ACTION Act_InitGlobal:

	(* Always Change If Project Change *)

	//Pass Data To Link
	p_bLinkOpsRun ACCESS p_OpsRun;
	p_bLinkOpsSimu ACCESS p_SimuRun;

	p_bLinkDISafetyRlySig ACCESS p_DISafetyRlySig;

	//Pass Data To Internal Use
	p_udiRstErr ACCESS p_RstErrReset;
	p_bPrep ACCESS p_NtParamProjInletShutPrep;
	p_bDis ACCESS p_McParamInShutterDis;
	p_bManual ACCESS p_UIMnlMod;
	p_bTwoCtrlIn ACCESS p_NtParamInShutterTwoCtrlIn;
	p_sProgNm ACCESS p_NtParamInShutterProgNm;
	p_bExtSen ACCESS p_DIInShutterCloseRS;
	p_bRetSen ACCESS p_DIInShutterOpenRS;
	p_tExtTO ACCESS p_NtParamInShutterExtTO;
	p_tRetTO ACCESS p_NtParamInShutterRetTO;
	p_bNtSettingsLoadDone ACCESS p_StartupNtSettingsLoadDone;

	(* Always Change If Project Change *)

END_ACTION
```

#### InputRef_Link.var - Change By Project
```iecst
(*2019-04-09*)
(**)
(*External*)
VAR
	p_bLinkOpsRun : REFERENCE TO BOOL;
END_VAR
(**)
VAR
	p_bLinkDISafetyRlySig : REFERENCE TO BOOL;
END_VAR
(**)
VAR
	p_bLinkOpsSimu : REFERENCE TO BOOL;
END_VAR
```

#### Act_LinkAction.st - Change By Project
```iecst
(** 2019-04-09 **)
ACTION Act_LinkAction:

	IF p_bLinkOpsRun = TRUE THEN
		p_eAct ACCESS p_OpsInvertInletShutterAct;
	ELSIF p_bLinkOpsSimu = TRUE THEN
		p_eAct ACCESS p_SimuInvInShutterAct;
	ELSIF p_bManual = TRUE THEN
		p_eAct ACCESS p_UIInShutterAct;
	ELSE
		p_eAct ACCESS ADR(eAct);
	END_IF

END_ACTION
```

#### Act_InitLocal.st - Do Not Change!!!
```iecst
(** 2019-03-25 **)
ACTION Act_InitLocal:

	//Input Reference Link To Local Variable
	p_eAct ACCESS ADR(eAct);
	p_udiRstErr ACCESS ADR(udiRstErr);
	p_bPrep ACCESS ADR(bPrep);
	p_bEn ACCESS ADR(bEn);
	p_bDis ACCESS ADR(bDis);
	p_bManual ACCESS ADR(bManual);
	p_bTwoCtrlIn ACCESS ADR(bTwoCtrlIn);
	p_bExtSafetySen ACCESS ADR(bExtSafetySen);
	p_bRetSafetySen ACCESS ADR(bRetSafetySen);
	p_sProgNm ACCESS ADR(sProgNm);
	p_tExtTO ACCESS ADR(tExtTO);
	p_tRetTO ACCESS ADR(tRetTO);
	p_bNtSettingsLoadDone ACCESS ADR(bNtSettingsLoadDone);
	p_bExtSen ACCESS ADR(bExtSen);
	p_bRetSen ACCESS ADR(bRetSen);

END_ACTION
```

#### Act_Initial.st - Do Not Change!!!
```iecst
(** 2019-03-22 **)
ACTION Act_Initial:

	//Initial
	sStatTxt	:= a_sStatText[eStat];

	bTwoCtrlOut	:= p_bTwoCtrlIn;

	fbPneuExtChk.tTimeOut	:= p_tExtTO;
	fbPneuExtChk(bEn := FALSE);

	fbPneuRetChk.tTimeOut	:= p_tRetTO;
	fbPneuRetChk(bEn := FALSE);

END_ACTION
```

#### Act_Background.st - Do Not Change!!!
```iecst
(** 2018-12-14 **)
ACTION Act_Background:

	IF p_bExtSen = FALSE THEN
		bExtended	:= FALSE;
	END_IF

	IF p_bRetSen = FALSE THEN
		bRetracted	:= FALSE;
	END_IF

END_ACTION
```

#### Act_Alarm.st - Do Not Change!!!
```iecst
(** 2019-03-25 **)
ACTION Act_Alarm:

	//Error
	IF EDGEPOS(eStatus = Error) THEN

		tyAlmData.sProgNm		:= p_sProgNm;
		tyAlmData.udiCode		:= udiStatus;
		tyAlmData.eSeverity		:= AlmSeverityError;
		tyAlmData.udiRunTime	:= tyAlmData.udiRunTime + 1;
		tyAlmData.bAlm			:= TRUE;
		tyAlmData.udiModuleNum  := udiModuleNum;
		g_sPneu2SenProgNm		:= p_sProgNm;

		//Get Error Message
		IF tyAlmData.udiCode < 10000 OR tyAlmData.udiCode > 10099 THEN
			tyAlmData.sAlmMsg	:= 'Unknown';
			tyAlmData.sRcyMsg	:= 'Unknown';
		ELSE
			tyAlmData.sAlmMsg	:= a_tyAlmText[tyAlmData.udiCode].sAlmText;
			tyAlmData.sRcyMsg	:= a_tyAlmText[tyAlmData.udiCode].sRcyText;
		END_IF

		sStatTxt	:= tyAlmData.sAlmMsg;

	ELSIF bRstErr AND (tyAlmData.udiCode <> 0) THEN

		tyAlmData.udiCode	:= 0;
		tyAlmData.eSeverity	:= AlmSeverityNA;
		tyAlmData.sAlmMsg	:= '';
		tyAlmData.sRcyMsg	:= '';
		tyAlmData.bAlm			:= FALSE;
		sStatTxt	:= a_sStatText[eStat];

	END_IF

END_ACTION
```

#### Local.var - Do Not Change!!!
```iecst
(*2019-04-30*)
(**)
(*Local Action, State & Status*)
VAR
	eAct : ePneuAction := PneuActIdle;
	eStat : ePneuAction := PneuActIdle;
	eStatus : eFBStatus := Idle;
	udiStatus : UDINT := 0;
	sStatTxt : STRING[200] := '';
	a_sStatText : ARRAY[0..50] OF STRING[200] := ['Idling','Set All','Reset All','Set Extend','Set Retract','Extending','Retracting','Retracting From Extend Sensor To Middle Sensor','Retracting From Middle Sensor To Retract Sensor','Extending From Retract Sensor To Middle Sensor','Extending From Middle Sensor To Extend Sensor',40('')];
END_VAR
(**)
(*Local Alarm*)
VAR
	tyAlmData : tyAlmDat;
	a_tyAlmText : ARRAY[10000..10099] OF tyAlmTxt := [(sAlmText:='Safety Check Error While Extending',sRcyText:='Safety System Has Been Triggered. All Operations Are Disable. Remove the Obstacle That Triggered The Safety Interlock To Resume Operation.'),(sAlmText:='Extend Sensor On Checking Time Out While Extending',sRcyText:='Sensor Timeout Expired Before Operation Completed. Sensor Operation Is Abnormal. Solve The Error To Resume Operation. '),(sAlmText:='Retract Sensor Off Checking Time Out While Extending',sRcyText:='Sensor Timeout Expired Before Operation Completed. Sensor Operation Is Abnormal. Solve The Error To Resume Operation.'),(sAlmText:='Safety Check Error While Retracting',sRcyText:='Safety System Has Been Triggered. All Operations Are Disable. Remove the Obstacle That Triggered The Safety Interlock To Resume Operation.'),(sAlmText:='Retract Sensor On Checking Time Out While Retracting',sRcyText:='Sensor Timeout Expired Before Operation Completed. Sensor Operation Is Abnormal. Solve The Error To Resume Operation.'),(sAlmText:='Extend Sensor Off Checking Time Out While Retracting',sRcyText:='Sensor Timeout Expired Before Operation Completed. Sensor Operation Is Abnormal. Solve The Error To Resume Operation.'),94((0))];
END_VAR
(**)
(*Local Output*)
VAR
	bExtCtrl : BOOL;
	bRetCtrl : BOOL;
	bTwoCtrlOut : BOOL := FALSE;
	bExtended : BOOL := FALSE;
	bRetracted : BOOL := FALSE;
END_VAR
(**)
(*Local Input*)
VAR
	udiRstErr : UDINT := 0;
	bPrep : BOOL := TRUE;
	bEn : BOOL := TRUE;
	bDis : BOOL := FALSE;
	bManual : BOOL := FALSE;
	bTwoCtrlIn : BOOL := FALSE;
	bExtSafetySen : BOOL := TRUE;
	bRetSafetySen : BOOL := TRUE;
	bExtSen : BOOL := FALSE;
	bRetSen : BOOL := FALSE;
	sProgNm : STRING[15] := 'Pneu2Sen';
	tExtTO : TIME := T#20s;
	tRetTO : TIME := T#20s;
	bNtSettingsLoadDone : BOOL := TRUE;
END_VAR
(**)
(*Local*)
VAR
	bRstErr : BOOL;
	udiRstErrOld : UDINT;
	bInitDone : BOOL;
	bInitialDone : BOOL;
	fbPneuExtChk : fbPneuExtRetSenExtChk;
	fbPneuRetChk : fbPneuExtRetSenRetChk;
	eStatOld : ePneuAction := PneuActIdle;
	udiModuleNum : UDINT := 2551;
END_VAR
```

### Pneu2SenOutShutter.var - Change By Project
```iecst
(*2019-03-25*)
(**)
(*Action & State & Status*)
VAR
	p_Pneu2SenOutShutterStat : UDINT;
	p_Pneu2SenOutShutterStatus : UDINT;
	p_Pneu2SenOutShutterStatTxt : UDINT;
END_VAR
(**)
(*Alarm*)
VAR
	p_Pneu2SenOutShutterAlmData : UDINT;
END_VAR
(**)
(*Output*)
VAR
	p_Pneu2SenOutShutterExtCtrl : UDINT;
	p_Pneu2SenOutShutterRetCtrl : UDINT;
	p_Pneu2SenOutShutterTwoCtrlOut : UDINT;
	p_Pneu2SenOutShutterExtended : UDINT;
	p_Pneu2SenOutShutterRetracted : UDINT;
END_VAR
```

### Program Logical/Pneu/Pneu2SenOutShutter (IEC) - 1.00.0 - NtPneu v5.00.0

#### InputRef.var
```iecst
(*2019-03-25*)
(**)
(*General*)
VAR
	p_eAct : REFERENCE TO ePneuAction;
	p_udiRstErr : REFERENCE TO UDINT;
	p_bPrep : REFERENCE TO BOOL;
	p_bEn : REFERENCE TO BOOL;
	p_bDis : REFERENCE TO BOOL;
END_VAR
(**)
(*Configuration*)
VAR
	p_bManual : REFERENCE TO BOOL;
	p_bTwoCtrlIn : REFERENCE TO BOOL;
	p_bExtSafetySen : REFERENCE TO BOOL;
	p_bRetSafetySen : REFERENCE TO BOOL;
	p_sProgNm : REFERENCE TO STRING[15];
	p_tExtTO : REFERENCE TO TIME;
	p_tRetTO : REFERENCE TO TIME;
	p_bNtSettingsLoadDone : REFERENCE TO BOOL;
END_VAR
(**)
(*Input*)
VAR
	p_bExtSen : REFERENCE TO BOOL;
	p_bRetSen : REFERENCE TO BOOL;
END_VAR
```

#### Act_InitGlobal.st
```iecst
(** 2019-04-09 **)
ACTION Act_InitGlobal:

	(* Always Change If Project Change *)

	//Pass Data To Link
	p_bLinkOpsRun ACCESS p_OpsRun;
	p_bLinkOpsSimu ACCESS p_SimuRun;

	p_bLinkDISafetyRlySig ACCESS p_DISafetyRlySig;

	//Pass Data To Internal Use
	p_udiRstErr ACCESS p_RstErrReset;
	p_bPrep ACCESS p_NtParamProjOutletShutPrep;
	p_bDis ACCESS p_McParamOutShutterDis;
	p_bManual ACCESS p_UIMnlMod;
	p_bTwoCtrlIn ACCESS p_NtParamOutShutterTwoCtrlIn;
	p_sProgNm ACCESS p_NtParamOutShutterProgNm;
	p_bExtSen ACCESS p_DIOutShutterCloseRS;
	p_bRetSen ACCESS p_DIOutShutterOpenRS;
	p_tExtTO ACCESS p_NtParamOutShutterExtTO;
	p_tRetTO ACCESS p_NtParamOutShutterRetTO;
	p_bNtSettingsLoadDone ACCESS p_StartupNtSettingsLoadDone;

	(* Always Change If Project Change *)

END_ACTION
```

#### Act_LinkAction.st
```iecst
(** 2019-04-09 **)
ACTION Act_LinkAction:

	IF p_bLinkOpsRun = TRUE THEN
		p_eAct ACCESS p_OpsInvertOutletShutterAct;
	ELSIF p_bLinkOpsSimu = TRUE THEN
		p_eAct ACCESS p_SimuInvOutShutterAct;
	ELSIF p_bManual = TRUE THEN
		p_eAct ACCESS p_UIOutShutterAct;
	ELSE
		p_eAct ACCESS ADR(eAct);
	END_IF

END_ACTION
```

#### Init.st
```iecst
(** 2019-03-25 **)
PROGRAM _INIT

	(* Always Change If Project Change *)

	//Pass Address To Global Address For External Use
	//Action, State & Status
	p_Pneu2SenOutShutterStat		:= ADR(eStat);
	p_Pneu2SenOutShutterStatus		:= ADR(eStatus);
	p_Pneu2SenOutShutterStatTxt		:= ADR(sStatTxt);

	//Alarm
	p_Pneu2SenOutShutterAlmData		:= ADR(tyAlmData);

	//Output
	p_Pneu2SenOutShutterExtCtrl		:= ADR(bExtCtrl);
	p_Pneu2SenOutShutterRetCtrl		:= ADR(bRetCtrl);
	p_Pneu2SenOutShutterTwoCtrlOut	:= ADR(bTwoCtrlOut);
	p_Pneu2SenOutShutterExtended	:= ADR(bExtended);
	p_Pneu2SenOutShutterRetracted	:= ADR(bRetracted);

	(* Always Change If Project Change *)

END_PROGRAM
```

### Pneu2SenClamp1.var - Change By Project
```iecst
(*2019-03-25*)
(**)
(*Action & State & Status*)
VAR
	p_Pneu2SenClamp1Stat : UDINT;
	p_Pneu2SenClamp1Status : UDINT;
	p_Pneu2SenClamp1StatTxt : UDINT;
END_VAR
(**)
(*Alarm*)
VAR
	p_Pneu2SenClamp1AlmData : UDINT;
END_VAR
(**)
(*Output*)
VAR
	p_Pneu2SenClamp1ExtCtrl : UDINT;
	p_Pneu2SenClamp1RetCtrl : UDINT;
	p_Pneu2SenClamp1TwoCtrlOut : UDINT;
	p_Pneu2SenClamp1Extended : UDINT;
	p_Pneu2SenClamp1Retracted : UDINT;
END_VAR
```

### Program Logical/Pneu/Pneu2SenInClamp1 (IEC) - 1.00.0 - NtPneu v5.00.0

#### InputRef.var
```iecst
(*2020-10-08*)
(**)
(*General*)
VAR
	p_eAct : REFERENCE TO ePneuAction;
	p_udiRstErr : REFERENCE TO UDINT;
	p_bPrep : REFERENCE TO BOOL;
	p_bEn : REFERENCE TO BOOL;
	p_bDis : REFERENCE TO BOOL;
END_VAR
(**)
(*Configuration*)
VAR
	p_bClampPrep : REFERENCE TO BOOL;
	p_eClampOption : REFERENCE TO eClampType;
	p_bManual : REFERENCE TO BOOL;
	p_bTwoCtrlIn : REFERENCE TO BOOL;
	p_bExtSafetySen : REFERENCE TO BOOL;
	p_bRetSafetySen : REFERENCE TO BOOL;
	p_sProgNm : REFERENCE TO STRING[15];
	p_tExtTO : REFERENCE TO TIME;
	p_tRetTO : REFERENCE TO TIME;
	p_bNtSettingsLoadDone : REFERENCE TO BOOL;
END_VAR
(**)
(*Input*)
VAR
	p_bExtSen : REFERENCE TO BOOL;
	p_bRetSen : REFERENCE TO BOOL;
END_VAR
```

#### Act_InitGlobal.st
```iecst
(** 2020-10-08 **)
ACTION Act_InitGlobal:

	(* Always Change If Project Change *)

	//Pass Data To Link
	p_bLinkOpsRun ACCESS p_OpsRun;

	p_bLinkDISafetyRlySig ACCESS p_DISafetyRlySig;

	//Pass Data To Internal Use
	p_udiRstErr ACCESS p_RstErrReset;
	p_bDis ACCESS p_McParamClampDis;
	p_bManual ACCESS p_UIMnlMod;
	p_bTwoCtrlIn ACCESS p_NtParamClamp1TwoCtrlIn;
	p_sProgNm ACCESS p_NtParamClamp1ProgNm;
	p_bExtSen ACCESS p_DIClampRS1;
	p_bRetSen ACCESS p_DIUnClampRS1;
	p_tExtTO ACCESS p_NtParamClamp1ExtTO;
	p_tRetTO ACCESS p_NtParamClamp1RetTO;
	p_bNtSettingsLoadDone ACCESS p_StartupNtSettingsLoadDone;

	p_bClampPrep ACCESS p_NtParamProjClampPrep;
	p_eClampOption ACCESS p_NtParamProjClampOption;

	(* Always Change If Project Change *)

END_ACTION
```

#### Act_LinkAction.st
```iecst
(** 2019-04-09 **)
ACTION Act_LinkAction:

	IF p_bLinkOpsRun = TRUE THEN
		p_eAct ACCESS p_OpsInvertClamp1Act;
	ELSIF p_bManual = TRUE THEN
		p_eAct ACCESS p_UIClamp1Act;
	ELSE
		p_eAct ACCESS ADR(eAct);
	END_IF

END_ACTION
```

#### Init.st
```iecst
(** 2019-03-25 **)
PROGRAM _INIT

	(* Always Change If Project Change *)

	//Pass Address To Global Address For External Use
	//Action, State & Status
	p_Pneu2SenClamp1Stat		:= ADR(eStat);
	p_Pneu2SenClamp1Status		:= ADR(eStatus);
	p_Pneu2SenClamp1StatTxt		:= ADR(sStatTxt);

	//Alarm
	p_Pneu2SenClamp1AlmData		:= ADR(tyAlmData);

	//Output
	p_Pneu2SenClamp1ExtCtrl		:= ADR(bExtCtrl);
	p_Pneu2SenClamp1RetCtrl		:= ADR(bRetCtrl);
	p_Pneu2SenClamp1TwoCtrlOut	:= ADR(bTwoCtrlOut);
	p_Pneu2SenClamp1Extended	:= ADR(bExtended);
	p_Pneu2SenClamp1Retracted	:= ADR(bRetracted);

	(* Always Change If Project Change *)

END_PROGRAM
```

### Pneu2SenClamp2.var - Change By Project
```iecst
(*2019-03-25*)
(**)
(*Action & State & Status*)
VAR
	p_Pneu2SenClamp2Stat : UDINT;
	p_Pneu2SenClamp2Status : UDINT;
	p_Pneu2SenClamp2StatTxt : UDINT;
END_VAR
(**)
(*Alarm*)
VAR
	p_Pneu2SenClamp2AlmData : UDINT;
END_VAR
(**)
(*Output*)
VAR
	p_Pneu2SenClamp2ExtCtrl : UDINT;
	p_Pneu2SenClamp2RetCtrl : UDINT;
	p_Pneu2SenClamp2TwoCtrlOut : UDINT;
	p_Pneu2SenClamp2Extended : UDINT;
	p_Pneu2SenClamp2Retracted : UDINT;
END_VAR
```

### Program Logical/Pneu/Pneu2SenInClamp2 (IEC) - 1.00.0 - NtPneu v5.00.0

#### Local.var
```iecst
(*2020-10-08*)
(**)
(*Local Action, State & Status*)
VAR
	eAct : ePneuAction := PneuActIdle;
	eStat : ePneuAction := PneuActIdle;
	eStatus : eFBStatus := Idle;
	udiStatus : UDINT := 0;
	sStatTxt : STRING[200] := '';
	a_sStatText : ARRAY[0..50] OF STRING[200] := ['Idling','Set All','Reset All','Set Extend','Set Retract','Extending','Retracting','Retracting From Extend Sensor To Middle Sensor','Retracting From Middle Sensor To Retract Sensor','Extending From Retract Sensor To Middle Sensor','Extending From Middle Sensor To Extend Sensor',40('')];
END_VAR
(**)
(*Local Alarm*)
VAR
	tyAlmData : tyAlmDat;
	a_tyAlmText : ARRAY[10000..10099] OF tyAlmTxt := [(sAlmText:='Safety Check Error While Extending',sRcyText:='Safety System Has Been Triggered. All Operations Are Disable. Remove the Obstacle That Triggered The Safety Interlock To Resume Operation.'),(sAlmText:='Extend Sensor On Checking Time Out While Extending',sRcyText:='Sensor Timeout Expired Before Operation Completed. Sensor Operation Is Abnormal. Solve The Error To Resume Operation. '),(sAlmText:='Retract Sensor Off Checking Time Out While Extending',sRcyText:='Sensor Timeout Expired Before Operation Completed. Sensor Operation Is Abnormal. Solve The Error To Resume Operation.'),(sAlmText:='Safety Check Error While Retracting',sRcyText:='Safety System Has Been Triggered. All Operations Are Disable. Remove the Obstacle That Triggered The Safety Interlock To Resume Operation.'),(sAlmText:='Retract Sensor On Checking Time Out While Retracting',sRcyText:='Sensor Timeout Expired Before Operation Completed. Sensor Operation Is Abnormal. Solve The Error To Resume Operation.'),(sAlmText:='Extend Sensor Off Checking Time Out While Retracting',sRcyText:='Sensor Timeout Expired Before Operation Completed. Sensor Operation Is Abnormal. Solve The Error To Resume Operation.'),94((0))];
END_VAR
(**)
(*Local Output*)
VAR
	bExtCtrl : BOOL;
	bRetCtrl : BOOL;
	bTwoCtrlOut : BOOL := FALSE;
	bExtended : BOOL := FALSE;
	bRetracted : BOOL := FALSE;
END_VAR
(**)
(*Local Input*)
VAR
	udiRstErr : UDINT := 0;
	bPrep : BOOL := TRUE;
	bEn : BOOL := TRUE;
	bDis : BOOL := FALSE;
	bClampPrep : BOOL := FALSE;
	eClampOption : eClampType := ClampNoRS;
	bManual : BOOL := FALSE;
	bTwoCtrlIn : BOOL := FALSE;
	bExtSafetySen : BOOL := TRUE;
	bRetSafetySen : BOOL := TRUE;
	bExtSen : BOOL := FALSE;
	bRetSen : BOOL := FALSE;
	sProgNm : STRING[15] := 'Pneu2Sen';
	tExtTO : TIME := T#20s;
	tRetTO : TIME := T#20s;
	bNtSettingsLoadDone : BOOL := TRUE;
END_VAR
(**)
(*Local*)
VAR
	bRstErr : BOOL;
	udiRstErrOld : UDINT;
	bInitDone : BOOL;
	bInitialDone : BOOL;
	fbPneuExtChk : fbPneuExtRetSenExtChk;
	fbPneuRetChk : fbPneuExtRetSenRetChk;
	eStatOld : ePneuAction := PneuActIdle;
	udiModuleNum : UDINT := 2551;
END_VAR
```

#### Act_Alarm.st
```iecst
(** 2019-03-25 **)
ACTION Act_Alarm:

	//Error
	IF EDGEPOS(eStatus = Error) THEN

		tyAlmData.sProgNm		:= p_sProgNm;
		tyAlmData.udiCode		:= udiStatus;
		tyAlmData.eSeverity		:= AlmSeverityError;
		tyAlmData.udiRunTime	:= tyAlmData.udiRunTime + 1;
		tyAlmData.bAlm			:= TRUE;
		tyAlmData.udiModuleNum  := udiModuleNum;
		g_sPneu2SenProgNm		:= p_sProgNm;

		//Get Error Message
		IF tyAlmData.udiCode < 10000 OR tyAlmData.udiCode > 10099 THEN
			tyAlmData.sAlmMsg	:= 'Unknown';
			tyAlmData.sRcyMsg	:= 'Unknown';
		ELSE
			tyAlmData.sAlmMsg	:= a_tyAlmText[tyAlmData.udiCode].sAlmText;
			tyAlmData.sRcyMsg	:= a_tyAlmText[tyAlmData.udiCode].sRcyText;
		END_IF

		sStatTxt	:= tyAlmData.sAlmMsg;

	ELSIF bRstErr AND (tyAlmData.udiCode <> 0) THEN

		tyAlmData.udiCode	:= 0;
		tyAlmData.eSeverity	:= AlmSeverityNA;
		tyAlmData.sAlmMsg	:= '';
		tyAlmData.sRcyMsg	:= '';
		tyAlmData.bAlm		:= FALSE;

		sStatTxt	:= a_sStatText[eStat];

	END_IF

END_ACTION
```

#### Act_InitGlobal.st
```iecst
(** 2020-10-08 **)
ACTION Act_InitGlobal:

	(* Always Change If Project Change *)

	//Pass Data To Link
	p_bLinkOpsRun ACCESS p_OpsRun;

	p_bLinkDISafetyRlySig ACCESS p_DISafetyRlySig;

	//Pass Data To Internal Use
	p_udiRstErr ACCESS p_RstErrReset;
	p_bDis ACCESS p_McParamClampDis;
	p_bManual ACCESS p_UIMnlMod;
	p_bTwoCtrlIn ACCESS p_NtParamClamp2TwoCtrlIn;
	p_sProgNm ACCESS p_NtParamClamp2ProgNm;
	p_bExtSen ACCESS p_DIClampRS2;
	p_bRetSen ACCESS p_DIUnClampRS2;
	p_tExtTO ACCESS p_NtParamClamp2ExtTO;
	p_tRetTO ACCESS p_NtParamClamp2RetTO;
	p_bNtSettingsLoadDone ACCESS p_StartupNtSettingsLoadDone;

	p_bClampPrep ACCESS p_NtParamProjClampPrep;
	p_eClampOption ACCESS p_NtParamProjClampOption;

	(* Always Change If Project Change *)

END_ACTION
```

#### Act_Link.st
```iecst
(** 2019-03-29 **)
ACTION Act_Link:

	IF p_bLinkDISafetyRlySig = FALSE THEN
		bExtCtrl	:= FALSE;
		bRetCtrl	:= FALSE;
		bExtended	:= FALSE;
		bRetracted	:= FALSE;
	END_IF

END_ACTION
```

#### Act_LinkAction.st
```iecst
(** 2019-04-09 **)
ACTION Act_LinkAction:

	IF p_bLinkOpsRun = TRUE THEN
		p_eAct ACCESS p_OpsInvertClamp2Act;
	ELSIF p_bManual = TRUE THEN
		p_eAct ACCESS p_UIClamp2Act;
	ELSE
		p_eAct ACCESS ADR(eAct);
	END_IF

END_ACTION
```

#### Act_LinkEn.st
```iecst
(** 2020-10-08 **)
ACTION Act_LinkEn:

	//Link bPrep, bEn & bDis
	p_bPrep := p_bClampPrep AND (p_eClampOption=ThreeClampsWithRS);
END_ACTION
```

#### Act_Main.st
```iecst
(** 2019-01-10 **)
ACTION Act_Main:

	IF eStatOld <> eStat THEN
		fbPneuExtChk(bEn := FALSE);
		fbPneuRetChk(bEn := FALSE);

		sStatTxt	:= a_sStatText[eStat];

		eStatOld	:= eStat;

		eStatus		:= Busy;
	END_IF

	//Main
	CASE eStat OF

		PneuActIdle:
			eStatus	:= Idle;

		PneuActSetAll:
			IF eStatus = Idle OR eStatus = Busy THEN

				//Reset
				fbPneuExtChk(bEn := FALSE);
				fbPneuRetChk(bEn := FALSE);

				bExtCtrl	:= TRUE;
				bRetCtrl	:= TRUE;

				eStatus	:= Done;

			END_IF

		PneuActRstAll:
			IF eStatus = Idle OR eStatus = Busy THEN

				//Reset
				fbPneuExtChk(bEn := FALSE);
				fbPneuRetChk(bEn := FALSE);

				bExtCtrl	:= FALSE;
				bRetCtrl	:= FALSE;

				eStatus	:= Done;

			END_IF

		PneuActSetExt:
			IF eStatus = Idle OR eStatus = Busy THEN

				//Reset
				fbPneuExtChk(bEn := FALSE);
				fbPneuRetChk(bEn := FALSE);

				bExtCtrl	:= TRUE;
				bRetCtrl	:= FALSE;

				bExtended	:= TRUE;

				eStatus	:= Done;

			END_IF

		PneuActSetRet:
			IF eStatus = Idle OR eStatus = Busy THEN

				//Reset
				fbPneuExtChk(bEn := FALSE);
				fbPneuRetChk(bEn := FALSE);

				bExtCtrl	:= FALSE;
				bRetCtrl	:= TRUE;

				bRetracted	:= TRUE;

				eStatus	:= Done;

			END_IF

		PneuActExt:
			IF eStatus = Idle OR eStatus = Busy THEN

				eStatus	:= Busy;

				//Reset
				fbPneuRetChk(bEn := FALSE);

				bExtCtrl	:= TRUE;
				bRetCtrl	:= FALSE;

				fbPneuExtChk.bExtSen	:= p_bExtSen;
				fbPneuExtChk.bRetSen	:= p_bRetSen;
				fbPneuExtChk.bExtSafety	:= p_bExtSafetySen;
				fbPneuExtChk(bEn := TRUE);

				IF fbPneuExtChk.udiStatus = 0 THEN
					bExtended	:= TRUE;
					eStatus		:= Done;
				ELSIF fbPneuExtChk.udiStatus < 65534 THEN
					IF p_bTwoCtrlIn = TRUE THEN
						bExtCtrl	:= FALSE;
						bRetCtrl	:= FALSE;
					ELSE
						bExtCtrl	:= FALSE;
						bRetCtrl	:= TRUE;
					END_IF

					eStatus		:= Error;

					IF fbPneuExtChk.udiStatus = 1507 THEN
						udiStatus	:= 10000;	//Safety Check Error While Extending
					ELSIF fbPneuExtChk.udiStatus = 1503 THEN
						udiStatus	:= 10001;	//Extend Sensor On Checking Time Out While Extending
					ELSIF fbPneuExtChk.udiStatus = 1506 THEN
						udiStatus	:= 10002;	//Retract Sensor Off Checking Time Out While Extending
					ELSE
						udiStatus	:= fbPneuExtChk.udiStatus;
					END_IF
				END_IF

			END_IF

		PneuActRet:
			IF eStatus = Idle OR eStatus = Busy THEN

				eStatus	:= Busy;

				//Reset
				fbPneuExtChk(bEn := FALSE);

				bExtCtrl	:= FALSE;
				bRetCtrl	:= TRUE;

				fbPneuRetChk.bExtSen	:= p_bExtSen;
				fbPneuRetChk.bRetSen	:= p_bRetSen;
				fbPneuRetChk.bRetSafety	:= p_bRetSafetySen;
				fbPneuRetChk(bEn := TRUE);

				IF fbPneuRetChk.udiStatus = 0 THEN
					bRetracted	:= TRUE;
					eStatus		:= Done;
				ELSIF fbPneuRetChk.udiStatus < 65534 THEN
					IF p_bTwoCtrlIn = TRUE THEN
						bExtCtrl	:= FALSE;
						bRetCtrl	:= FALSE;
					ELSE
						bExtCtrl	:= TRUE;
						bRetCtrl	:= FALSE;
					END_IF

					eStatus		:= Error;

					IF fbPneuRetChk.udiStatus = 1508 THEN
						udiStatus	:= 10003;	//Safety Check Error While Retracting
					ELSIF fbPneuRetChk.udiStatus = 1505 THEN
						udiStatus	:= 10004;	//Retract Sensor On Checking Time Out While Retracting
					ELSIF fbPneuRetChk.udiStatus = 1504 THEN
						udiStatus	:= 10005;	//Extend Sensor Off Checking Time Out While Retracting
					ELSE
						udiStatus	:= fbPneuRetChk.udiStatus;
					END_IF
				END_IF

			END_IF

		ELSE
			IF eStatus = Idle OR eStatus = Busy THEN
				eStatus	:= Done;
			END_IF

	END_CASE

END_ACTION
```

#### Init.st
```iecst
(** 2019-03-25 **)
PROGRAM _INIT

	(* Always Change If Project Change *)

	//Pass Address To Global Address For External Use
	//Action, State & Status
	p_Pneu2SenClamp2Stat		:= ADR(eStat);
	p_Pneu2SenClamp2Status		:= ADR(eStatus);
	p_Pneu2SenClamp2StatTxt		:= ADR(sStatTxt);

	//Alarm
	p_Pneu2SenClamp2AlmData		:= ADR(tyAlmData);

	//Output
	p_Pneu2SenClamp2ExtCtrl		:= ADR(bExtCtrl);
	p_Pneu2SenClamp2RetCtrl		:= ADR(bRetCtrl);
	p_Pneu2SenClamp2TwoCtrlOut	:= ADR(bTwoCtrlOut);
	p_Pneu2SenClamp2Extended	:= ADR(bExtended);
	p_Pneu2SenClamp2Retracted	:= ADR(bRetracted);

	(* Always Change If Project Change *)

END_PROGRAM
```

### Pneu2SenClamp3.var - Change By Project
```iecst
(*2019-03-25*)
(**)
(*Action & State & Status*)
VAR
	p_Pneu2SenClamp3Stat : UDINT;
	p_Pneu2SenClamp3Status : UDINT;
	p_Pneu2SenClamp3StatTxt : UDINT;
END_VAR
(**)
(*Alarm*)
VAR
	p_Pneu2SenClamp3AlmData : UDINT;
END_VAR
(**)
(*Output*)
VAR
	p_Pneu2SenClamp3ExtCtrl : UDINT;
	p_Pneu2SenClamp3RetCtrl : UDINT;
	p_Pneu2SenClamp3TwoCtrlOut : UDINT;
	p_Pneu2SenClamp3Extended : UDINT;
	p_Pneu2SenClamp3Retracted : UDINT;
END_VAR
```

### Program Logical/Pneu/Pneu2SenInClamp3 (IEC) - 1.00.0 - NtPneu v5.00.0

#### Act_Action.st
```iecst
(** 2019-03-25 **)
ACTION Act_Action:

	//Reset Error
	IF (eStatus = Error) AND bRstErr THEN
		p_eAct	:= PneuActIdle;
		eStat	:= PneuActIdle;
	END_IF

	//Set p_eAct
	IF eStatus = Idle OR eStatus = Busy OR eStatus = Done THEN
		eStat	:= p_eAct;
	END_IF

END_ACTION
```

#### Act_InitGlobal.st
```iecst
(** 2020-10-08 **)
ACTION Act_InitGlobal:

	(* Always Change If Project Change *)

	//Pass Data To Link
	p_bLinkOpsRun ACCESS p_OpsRun;

	p_bLinkDISafetyRlySig ACCESS p_DISafetyRlySig;

	//Pass Data To Internal Use
	p_udiRstErr ACCESS p_RstErrReset;
	p_bDis ACCESS p_McParamClampDis;
	p_bManual ACCESS p_UIMnlMod;
	p_bTwoCtrlIn ACCESS p_NtParamClamp3TwoCtrlIn;
	p_sProgNm ACCESS p_NtParamClamp3ProgNm;
	p_bExtSen ACCESS p_DIClampRS3;
	p_bRetSen ACCESS p_DIUnClampRS3;
	p_tExtTO ACCESS p_NtParamClamp3ExtTO;
	p_tRetTO ACCESS p_NtParamClamp3RetTO;
	p_bNtSettingsLoadDone ACCESS p_StartupNtSettingsLoadDone;

	p_bClampPrep ACCESS p_NtParamProjClampPrep;
	p_eClampOption ACCESS p_NtParamProjClampOption;
	(* Always Change If Project Change *)

END_ACTION
```

#### Act_InitLocal.st
```iecst
(** 2020-10-08 **)
ACTION Act_InitLocal:

	//Input Reference Link To Local Variable
	p_eAct ACCESS ADR(eAct);
	p_udiRstErr ACCESS ADR(udiRstErr);
	p_bPrep ACCESS ADR(bPrep);
	p_bEn ACCESS ADR(bEn);
	p_bDis ACCESS ADR(bDis);
	p_bClampPrep ACCESS ADR(bClampPrep);
	p_eClampOption ACCESS ADR(eClampOption);
	p_bManual ACCESS ADR(bManual);
	p_bTwoCtrlIn ACCESS ADR(bTwoCtrlIn);
	p_bExtSafetySen ACCESS ADR(bExtSafetySen);
	p_bRetSafetySen ACCESS ADR(bRetSafetySen);
	p_sProgNm ACCESS ADR(sProgNm);
	p_tExtTO ACCESS ADR(tExtTO);
	p_tRetTO ACCESS ADR(tRetTO);
	p_bNtSettingsLoadDone ACCESS ADR(bNtSettingsLoadDone);
	p_bExtSen ACCESS ADR(bExtSen);
	p_bRetSen ACCESS ADR(bRetSen);

END_ACTION
```

#### Act_LinkAction.st
```iecst
(** 2019-04-09 **)
ACTION Act_LinkAction:

	IF p_bLinkOpsRun = TRUE THEN
	p_eAct ACCESS p_OpsInvertClamp3Act;
	ELSIF p_bManual = TRUE THEN
		p_eAct ACCESS p_UIClamp3Act;
	ELSE
		p_eAct ACCESS ADR(eAct);
	END_IF

END_ACTION
```

#### Cyclic.st
```iecst
(** 2019-03-29 **)
PROGRAM _CYCLIC

	IF bInitDone = FALSE THEN
		bInitDone	:= TRUE;

		Act_InitLocal;
		Act_InitGlobal;

	ELSIF bInitialDone = FALSE THEN
		IF p_bNtSettingsLoadDone = TRUE THEN
			bInitialDone	:= TRUE;

			Act_Initial;
		END_IF

	ELSE

		Act_RstErr;
		Act_LinkAction;
		Act_Action;
		Act_LinkEn;

		IF (p_bPrep = TRUE) AND (p_bEn = TRUE) AND (p_bDis = FALSE) THEN
			Act_Link;
			Act_Main;
			Act_Background;
		ELSE
			IF eStat <> PneuActIdle THEN
				IF eStat = PneuActSetExt OR eStat = PneuActExt THEN
					bExtended	:= TRUE;
					bRetracted	:= FALSE;
				ELSIF eStat = PneuActSetRet OR eStat = PneuActRet THEN
					bExtended	:= FALSE;
					bRetracted	:= TRUE;
				END_IF

				eStatus	:= Done;
			ELSE
				eStatus	:= Idle;
			END_IF
		END_IF

		Act_Alarm;

	END_IF

END_PROGRAM
```

#### Init.st
```iecst
(** 2019-03-25 **)
PROGRAM _INIT

	(* Always Change If Project Change *)

	//Pass Address To Global Address For External Use
	//Action, State & Status
	p_Pneu2SenClamp3Stat		:= ADR(eStat);
	p_Pneu2SenClamp3Status		:= ADR(eStatus);
	p_Pneu2SenClamp3StatTxt		:= ADR(sStatTxt);

	//Alarm
	p_Pneu2SenClamp3AlmData		:= ADR(tyAlmData);

	//Output
	p_Pneu2SenClamp3ExtCtrl		:= ADR(bExtCtrl);
	p_Pneu2SenClamp3RetCtrl		:= ADR(bRetCtrl);
	p_Pneu2SenClamp3TwoCtrlOut	:= ADR(bTwoCtrlOut);
	p_Pneu2SenClamp3Extended	:= ADR(bExtended);
	p_Pneu2SenClamp3Retracted	:= ADR(bRetracted);

	(* Always Change If Project Change *)

END_PROGRAM
```

### Conv.typ - Change By Project
```iecst
(*2019-06-17*)
(**)
(*Action*)

TYPE
	eConvAction :
		(
		ConvActIdle,
		ConvActInit,
		ConvActInitRev,
		ConvActInitPshr,
		ConvActInitPuller,
		ConvActInitRej,
		ConvActInitInsp,
		ConvActEnt,
		ConvActEntToInOff,
		ConvActEntRev,
		ConvActRev,
		ConvActRevImmedStart,
		ConvActEntPuller,
		ConvActEntRej,
		ConvActEntInsp,
		ConvActPreExit,
		ConvActRejResume,
		ConvActExit,
		ConvActExit1,
		ConvActExitPshr,
		ConvActExit1Pshr,
		ConvActPshrSetAll,
		ConvActPshrRstAll,
		ConvActPshrSetExt,
		ConvActPshrSetRet,
		ConvActPshrExt,
		ConvActPshrRet,
		ConvActPullerSetAll,
		ConvActPullerRstAll,
		ConvActPullerSetExt,
		ConvActPullerSetRet,
		ConvActPullerExt,
		ConvActPullerRet,
		ConvActRotSetAll,
		ConvActRotRstAll,
		ConvActRotSetHome,
		ConvActRotSetRmt,
		ConvActRotHome,
		ConvActRotRemote,
		ConvActRejSetAll,
		ConvActRejRstAll,
		ConvActRejSetUp,
		ConvActRejSetDown,
		ConvActRejUp,
		ConvActRejDown,
		ConvActStop,
		ConvActStopPshr,
		ConvActStopPuller,
		ConvActStopRej,
		ConvActSetMtrSigOnOrLToR,
		ConvActSetMtrDirOrRToL,
		ConvActRstMtrSigOnOrLToR,
		ConvActRstMtrDirOrRToL,
		ConvActSetMtrAll,
		ConvActRstMtrAll
		);
END_TYPE

(**)

TYPE
	eConvDir :
		(
		ConvDirLToR,
		ConvDirRToL,
		ConvDirLToL,
		ConvDirRToR
		);
END_TYPE
```

### Conv.var - Change By Project
```iecst
(*2019-03-25*)
(**)
(*Action & State & Status*)
VAR
	p_ConvStat : UDINT;
	p_ConvStatus : UDINT;
	p_ConvStatTxt : UDINT;
END_VAR
(**)
(*Alarm*)
VAR
	p_ConvAlmData : UDINT;
END_VAR
(**)
(*Output*)
VAR
	p_ConvHvBrd : UDINT;
	p_ConvRejHvBrd : UDINT;
	p_ConvInspHvBrd : UDINT;
	p_ConvGdBrd : UDINT;
	p_ConvLmtSenActivated : UDINT;
	p_ConvMtrSigOnOrLToR : UDINT;
	p_ConvMtrDirOrRToL : UDINT;
	p_ConvPshrExtCtrl : UDINT;
	p_ConvPshrTwoOutputControl : UDINT;
	p_ConvPshrExtended : UDINT;
	p_ConvPshrRetracted : UDINT;
	p_ConvPullerExtCtrl : UDINT;
	p_ConvPullerRetCtrl : UDINT;
	p_ConvPullerTwoOutputControl : UDINT;
	p_ConvPullerExtended : UDINT;
	p_ConvPullerRetracted : UDINT;
	p_ConvRotRemoteCtrl : UDINT;
	p_ConvRotTwoOutputControl : UDINT;
	p_ConvRotAtRemote : UDINT;
	p_ConvRotAtHome : UDINT;
	p_ConvRejectUpCtrl : UDINT;
	p_ConvRejectDownCtrl : UDINT;
	p_ConvRejectTwoOutputControl : UDINT;
	p_ConvRejectAtUp : UDINT;
	p_ConvRejectAtDown : UDINT;
END_VAR
```

### Program Logical/Conv/Conv (IEC) - 1.00.0 - NtConv v5.00.0 , NtPneu v5.00.0

#### InputRef.var
```iecst
(*2019-03-25*)
(**)
(*General*)
VAR
	p_eAct : REFERENCE TO eConvAction;
	p_udiRstErr : REFERENCE TO UDINT;
	p_bPrep : REFERENCE TO BOOL;
	p_bEn : REFERENCE TO BOOL;
	p_bDis : REFERENCE TO BOOL;
END_VAR
(**)
(*Configuration*)
VAR
	p_bManual : REFERENCE TO BOOL;
	p_bLongBrdPrep : REFERENCE TO BOOL;
	p_bLongBrdEn : REFERENCE TO BOOL;
	p_bOnDirMod : REFERENCE TO BOOL;
	p_diInitTm : REFERENCE TO DINT;
	p_diRevDlyTm : REFERENCE TO DINT;
	p_tMtrOffDlyTm : REFERENCE TO TIME;
	p_diTxInTimeOut : REFERENCE TO DINT;
	p_diTxOutTimeOut : REFERENCE TO DINT;
	p_eDirection : REFERENCE TO eConvDir;
	p_bGdBrdInit : REFERENCE TO BOOL;
	p_bGdBrdEnt : REFERENCE TO BOOL;
	p_sProgNm : REFERENCE TO STRING[15];
	p_tPshrExtTO : REFERENCE TO TIME;
	p_tPshrRetTO : REFERENCE TO TIME;
	p_tPullerExtTO : REFERENCE TO TIME;
	p_tPullerRetTO : REFERENCE TO TIME;
	p_tRotHomeTO : REFERENCE TO TIME;
	p_tRotRemoteTO : REFERENCE TO TIME;
	p_tRejectUpTO : REFERENCE TO TIME;
	p_tRejectDownTO : REFERENCE TO TIME;
	p_bNtSettingsLoadDone : REFERENCE TO BOOL;
END_VAR
(**)
(*Input*)
VAR
	p_bLeftSen : REFERENCE TO BOOL;
	p_bRightSen : REFERENCE TO BOOL;
	p_bMiddleSen : REFERENCE TO BOOL;
	p_bPullerChkSen : REFERENCE TO BOOL;
	p_bPshrExtSen : REFERENCE TO BOOL;
	p_bPshrRetSen : REFERENCE TO BOOL;
	p_bPshrExtSafetySen : REFERENCE TO BOOL;
	p_bPshrRetSafetySen : REFERENCE TO BOOL;
	p_bPullerExtSen : REFERENCE TO BOOL;
	p_bPullerRetSen : REFERENCE TO BOOL;
	p_bPullerExtSafetySen : REFERENCE TO BOOL;
	p_bPullerRetSafetySen : REFERENCE TO BOOL;
	p_bRotHomeSen : REFERENCE TO BOOL;
	p_bRotRemoteSen : REFERENCE TO BOOL;
	p_bRotHomeSafetySen : REFERENCE TO BOOL;
	p_bRotRemoteSafetySen : REFERENCE TO BOOL;
	p_bRejectUpSen : REFERENCE TO BOOL;
	p_bRejectDownSen : REFERENCE TO BOOL;
	p_bRejectUpSafetySen : REFERENCE TO BOOL;
	p_bRejectDownSafetySen : REFERENCE TO BOOL;
	p_bUSHermesDSRdy : REFERENCE TO BOOL;
	p_bDSHermesUSRdy : REFERENCE TO BOOL;
	p_bUSHermesReversalDSRdy : REFERENCE TO BOOL;
	p_bDSHermesReversalUSRdy : REFERENCE TO BOOL;
END_VAR
```

#### InputRef_Link.var
```iecst
(*2019-04-09*)
(**)
VAR
	p_bLinkOpsRun : REFERENCE TO BOOL;
	p_bLinkOpsSimu : REFERENCE TO BOOL;
END_VAR
(**)
VAR
	p_bLinkUIBypsInitConv : REFERENCE TO BOOL;
	p_eLinkMcParamUSCommMod : REFERENCE TO eMcSetCommMod;
	p_bLinkOpsInvertBrdInserted : REFERENCE TO BOOL;
	p_eLinkMcParamUSComm2Mod : REFERENCE TO eMcSetCommMod;
	p_tyNtParamCurr : REFERENCE TO tyNtParam;
	p_bLinkOpsInvertOnceTwicePCBOut : REFERENCE TO BOOL;
	p_usiLinkMcMod : REFERENCE TO USINT;
	New_Variable : USINT;
END_VAR
```
